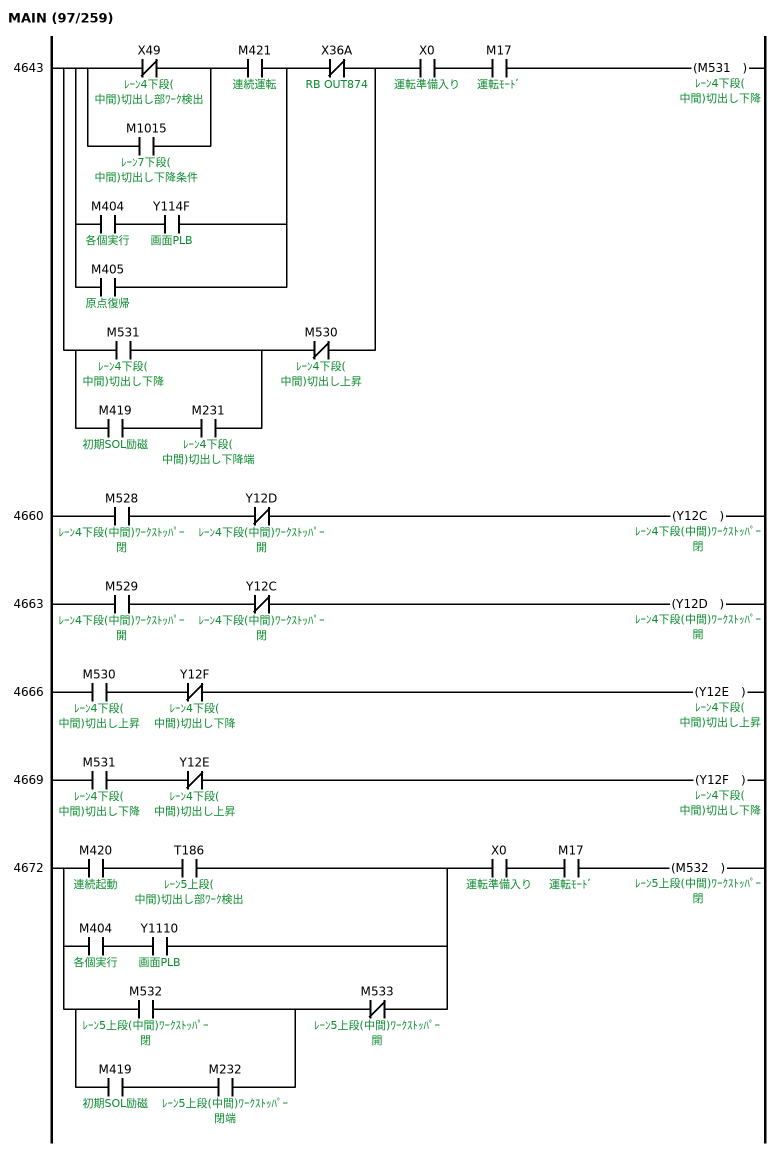
[picture p96: ladder of MAIN, rungs at steps 4643 to 4672]
4643  LDI     X49  ; ﾚｰﾝ4下段(中間)切出し部ﾜｰｸ検出
      OR      M1015  ; ﾚｰﾝ7下段(中間)切出し下降条件
      AND     M421  ; 連続運転
      LD      M404  ; 各個実行
      AND     Y114F  ; 画面PLB
      ORB
      OR      M405  ; 原点復帰
      ANI     X36A  ; RB OUT874
      LD      M531  ; ﾚｰﾝ4下段(中間)切出し下降
      LD      M419  ; 初期SOL励磁
      AND     M231  ; ﾚｰﾝ4下段(中間)切出し下降端
      ORB
      ANI     M530  ; ﾚｰﾝ4下段(中間)切出し上昇
      ORB
      AND     X0  ; 運転準備入り
      AND     M17  ; 運転ﾓｰﾄﾞ
      OUT     M531  ; ﾚｰﾝ4下段(中間)切出し下降
4660  LD      M528  ; ﾚｰﾝ4下段(中間)ﾜｰｸｽﾄｯﾊﾟｰ閉
      ANI     Y12D  ; ﾚｰﾝ4下段(中間)ﾜｰｸｽﾄｯﾊﾟｰ開
      OUT     Y12C  ; ﾚｰﾝ4下段(中間)ﾜｰｸｽﾄｯﾊﾟｰ閉
4663  LD      M529  ; ﾚｰﾝ4下段(中間)ﾜｰｸｽﾄｯﾊﾟｰ開
      ANI     Y12C  ; ﾚｰﾝ4下段(中間)ﾜｰｸｽﾄｯﾊﾟｰ閉
      OUT     Y12D  ; ﾚｰﾝ4下段(中間)ﾜｰｸｽﾄｯﾊﾟｰ開
4666  LD      M530  ; ﾚｰﾝ4下段(中間)切出し上昇
      ANI     Y12F  ; ﾚｰﾝ4下段(中間)切出し下降
      OUT     Y12E  ; ﾚｰﾝ4下段(中間)切出し上昇
4669  LD      M531  ; ﾚｰﾝ4下段(中間)切出し下降
      ANI     Y12E  ; ﾚｰﾝ4下段(中間)切出し上昇
      OUT     Y12F  ; ﾚｰﾝ4下段(中間)切出し下降
4672  LD      M420  ; 連続起動
      AND     T186  ; ﾚｰﾝ5上段(中間)切出し部ﾜｰｸ検出
      LD      M404  ; 各個実行
      AND     Y1110  ; 画面PLB
      ORB
      LD      M532  ; ﾚｰﾝ5上段(中間)ﾜｰｸｽﾄｯﾊﾟｰ閉
      LD      M419  ; 初期SOL励磁
      AND     M232  ; ﾚｰﾝ5上段(中間)ﾜｰｸｽﾄｯﾊﾟｰ閉端
      ORB
      ANI     M533  ; ﾚｰﾝ5上段(中間)ﾜｰｸｽﾄｯﾊﾟｰ開
      ORB
      AND     X0  ; 運転準備入り
      AND     M17  ; 運転ﾓｰﾄﾞ
      OUT     M532  ; ﾚｰﾝ5上段(中間)ﾜｰｸｽﾄｯﾊﾟｰ閉
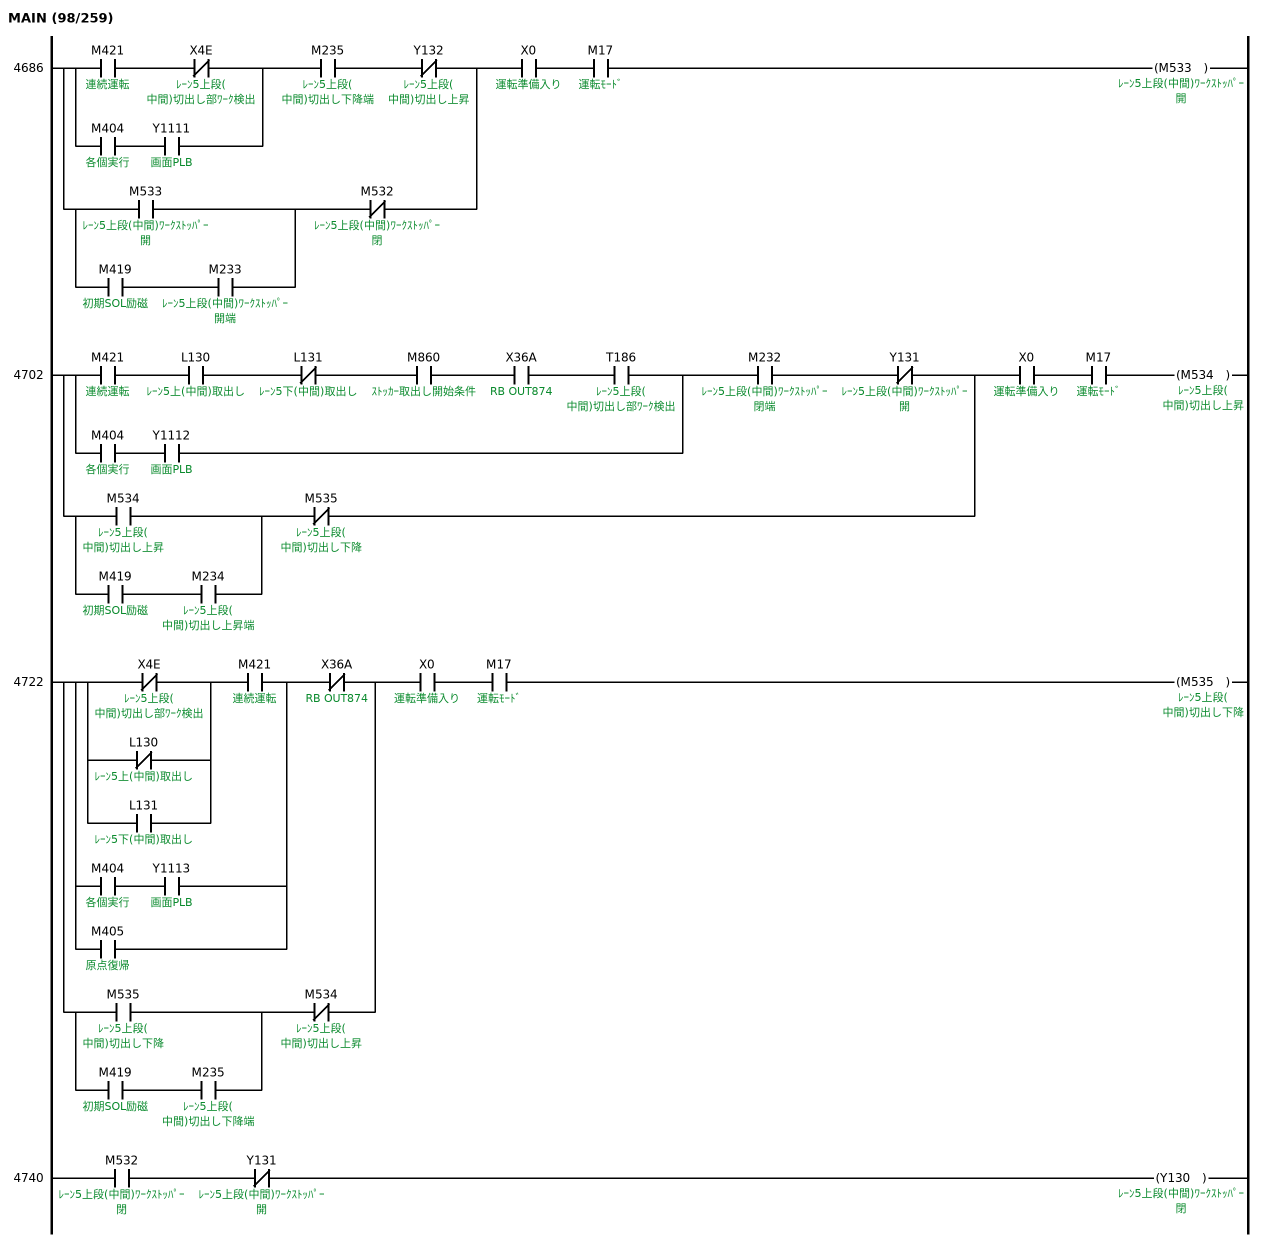
4686  LD      M421  ; 連続運転
      ANI     X4E  ; ﾚｰﾝ5上段(中間)切出し部ﾜｰｸ検出
      LD      M404  ; 各個実行
      AND     Y1111  ; 画面PLB
      ORB
      AND     M235  ; ﾚｰﾝ5上段(中間)切出し下降端
      ANI     Y132  ; ﾚｰﾝ5上段(中間)切出し上昇
      LD      M533  ; ﾚｰﾝ5上段(中間)ﾜｰｸｽﾄｯﾊﾟｰ開
      LD      M419  ; 初期SOL励磁
      AND     M233  ; ﾚｰﾝ5上段(中間)ﾜｰｸｽﾄｯﾊﾟｰ開端
      ORB
      ANI     M532  ; ﾚｰﾝ5上段(中間)ﾜｰｸｽﾄｯﾊﾟｰ閉
      ORB
      AND     X0  ; 運転準備入り
      AND     M17  ; 運転ﾓｰﾄﾞ
      OUT     M533  ; ﾚｰﾝ5上段(中間)ﾜｰｸｽﾄｯﾊﾟｰ開
4702  LD      M421  ; 連続運転
      AND     L130  ; ﾚｰﾝ5上(中間)取出し
      ANI     L131  ; ﾚｰﾝ5下(中間)取出し
      AND     M860  ; ｽﾄｯｶｰ取出し開始条件
      AND     X36A  ; RB OUT874
      AND     T186  ; ﾚｰﾝ5上段(中間)切出し部ﾜｰｸ検出
      LD      M404  ; 各個実行
      AND     Y1112  ; 画面PLB
      ORB
      AND     M232  ; ﾚｰﾝ5上段(中間)ﾜｰｸｽﾄｯﾊﾟｰ閉端
      ANI     Y131  ; ﾚｰﾝ5上段(中間)ﾜｰｸｽﾄｯﾊﾟｰ開
      LD      M534  ; ﾚｰﾝ5上段(中間)切出し上昇
      LD      M419  ; 初期SOL励磁
      AND     M234  ; ﾚｰﾝ5上段(中間)切出し上昇端
      ORB
      ANI     M535  ; ﾚｰﾝ5上段(中間)切出し下降
      ORB
      AND     X0  ; 運転準備入り
      AND     M17  ; 運転ﾓｰﾄﾞ
      OUT     M534  ; ﾚｰﾝ5上段(中間)切出し上昇
4722  LDI     X4E  ; ﾚｰﾝ5上段(中間)切出し部ﾜｰｸ検出
      ORI     L130  ; ﾚｰﾝ5上(中間)取出し
      OR      L131  ; ﾚｰﾝ5下(中間)取出し
      AND     M421  ; 連続運転
      LD      M404  ; 各個実行
      AND     Y1113  ; 画面PLB
      ORB
      OR      M405  ; 原点復帰
      ANI     X36A  ; RB OUT874
      LD      M535  ; ﾚｰﾝ5上段(中間)切出し下降
      LD      M419  ; 初期SOL励磁
      AND     M235  ; ﾚｰﾝ5上段(中間)切出し下降端
      ORB
      ANI     M534  ; ﾚｰﾝ5上段(中間)切出し上昇
      ORB
      AND     X0  ; 運転準備入り
      AND     M17  ; 運転ﾓｰﾄﾞ
      OUT     M535  ; ﾚｰﾝ5上段(中間)切出し下降
4740  LD      M532  ; ﾚｰﾝ5上段(中間)ﾜｰｸｽﾄｯﾊﾟｰ閉
      ANI     Y131  ; ﾚｰﾝ5上段(中間)ﾜｰｸｽﾄｯﾊﾟｰ開
      OUT     Y130  ; ﾚｰﾝ5上段(中間)ﾜｰｸｽﾄｯﾊﾟｰ閉
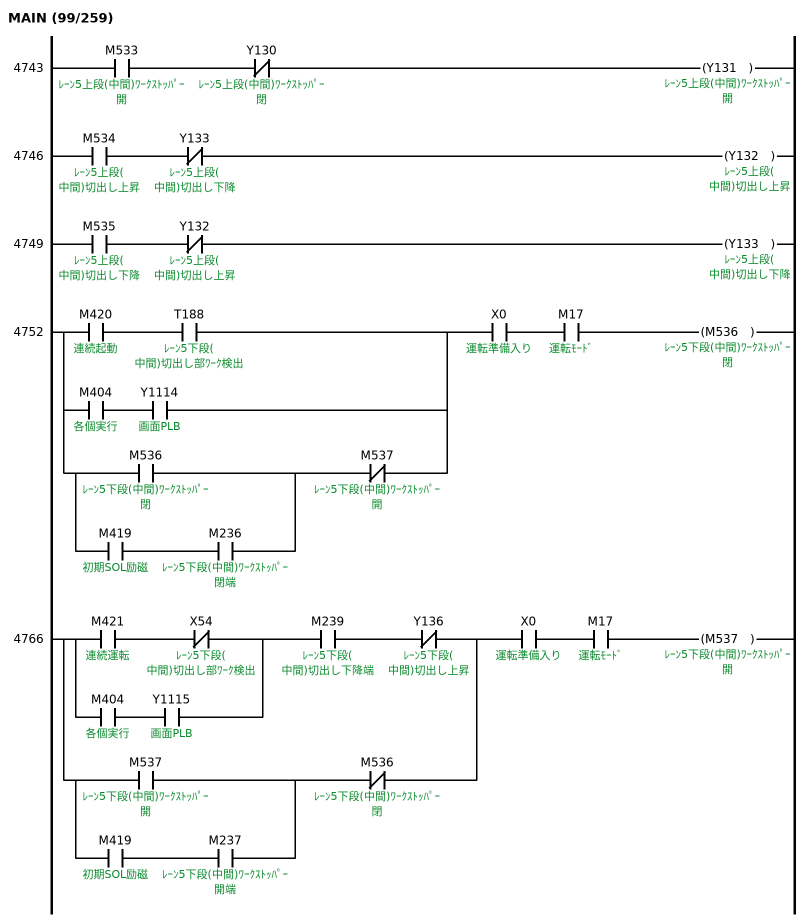
4743  LD      M533  ; ﾚｰﾝ5上段(中間)ﾜｰｸｽﾄｯﾊﾟｰ開
      ANI     Y130  ; ﾚｰﾝ5上段(中間)ﾜｰｸｽﾄｯﾊﾟｰ閉
      OUT     Y131  ; ﾚｰﾝ5上段(中間)ﾜｰｸｽﾄｯﾊﾟｰ開
4746  LD      M534  ; ﾚｰﾝ5上段(中間)切出し上昇
      ANI     Y133  ; ﾚｰﾝ5上段(中間)切出し下降
      OUT     Y132  ; ﾚｰﾝ5上段(中間)切出し上昇
4749  LD      M535  ; ﾚｰﾝ5上段(中間)切出し下降
      ANI     Y132  ; ﾚｰﾝ5上段(中間)切出し上昇
      OUT     Y133  ; ﾚｰﾝ5上段(中間)切出し下降
4752  LD      M420  ; 連続起動
      AND     T188  ; ﾚｰﾝ5下段(中間)切出し部ﾜｰｸ検出
      LD      M404  ; 各個実行
      AND     Y1114  ; 画面PLB
      ORB
      LD      M536  ; ﾚｰﾝ5下段(中間)ﾜｰｸｽﾄｯﾊﾟｰ閉
      LD      M419  ; 初期SOL励磁
      AND     M236  ; ﾚｰﾝ5下段(中間)ﾜｰｸｽﾄｯﾊﾟｰ閉端
      ORB
      ANI     M537  ; ﾚｰﾝ5下段(中間)ﾜｰｸｽﾄｯﾊﾟｰ開
      ORB
      AND     X0  ; 運転準備入り
      AND     M17  ; 運転ﾓｰﾄﾞ
      OUT     M536  ; ﾚｰﾝ5下段(中間)ﾜｰｸｽﾄｯﾊﾟｰ閉
4766  LD      M421  ; 連続運転
      ANI     X54  ; ﾚｰﾝ5下段(中間)切出し部ﾜｰｸ検出
      LD      M404  ; 各個実行
      AND     Y1115  ; 画面PLB
      ORB
      AND     M239  ; ﾚｰﾝ5下段(中間)切出し下降端
      ANI     Y136  ; ﾚｰﾝ5下段(中間)切出し上昇
      LD      M537  ; ﾚｰﾝ5下段(中間)ﾜｰｸｽﾄｯﾊﾟｰ開
      LD      M419  ; 初期SOL励磁
      AND     M237  ; ﾚｰﾝ5下段(中間)ﾜｰｸｽﾄｯﾊﾟｰ開端
      ORB
      ANI     M536  ; ﾚｰﾝ5下段(中間)ﾜｰｸｽﾄｯﾊﾟｰ閉
      ORB
      AND     X0  ; 運転準備入り
      AND     M17  ; 運転ﾓｰﾄﾞ
      OUT     M537  ; ﾚｰﾝ5下段(中間)ﾜｰｸｽﾄｯﾊﾟｰ開
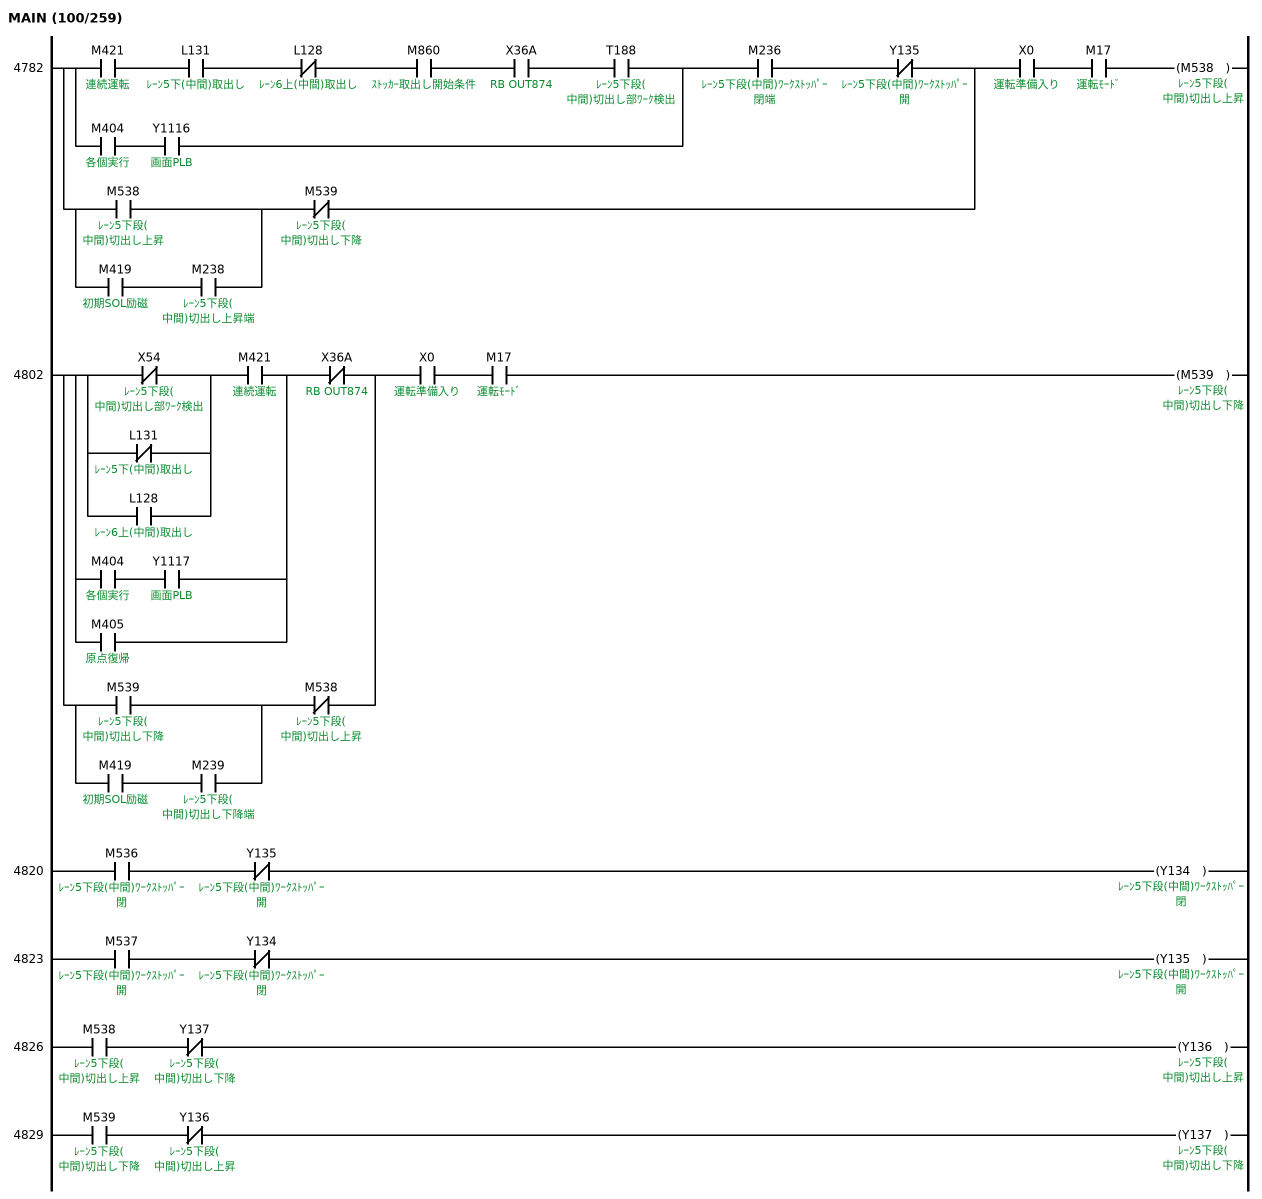
4782  LD      M421  ; 連続運転
      AND     L131  ; ﾚｰﾝ5下(中間)取出し
      ANI     L128  ; ﾚｰﾝ6上(中間)取出し
      AND     M860  ; ｽﾄｯｶｰ取出し開始条件
      AND     X36A  ; RB OUT874
      AND     T188  ; ﾚｰﾝ5下段(中間)切出し部ﾜｰｸ検出
      LD      M404  ; 各個実行
      AND     Y1116  ; 画面PLB
      ORB
      AND     M236  ; ﾚｰﾝ5下段(中間)ﾜｰｸｽﾄｯﾊﾟｰ閉端
      ANI     Y135  ; ﾚｰﾝ5下段(中間)ﾜｰｸｽﾄｯﾊﾟｰ開
      LD      M538  ; ﾚｰﾝ5下段(中間)切出し上昇
      LD      M419  ; 初期SOL励磁
      AND     M238  ; ﾚｰﾝ5下段(中間)切出し上昇端
      ORB
      ANI     M539  ; ﾚｰﾝ5下段(中間)切出し下降
      ORB
      AND     X0  ; 運転準備入り
      AND     M17  ; 運転ﾓｰﾄﾞ
      OUT     M538  ; ﾚｰﾝ5下段(中間)切出し上昇
4802  LDI     X54  ; ﾚｰﾝ5下段(中間)切出し部ﾜｰｸ検出
      ORI     L131  ; ﾚｰﾝ5下(中間)取出し
      OR      L128  ; ﾚｰﾝ6上(中間)取出し
      AND     M421  ; 連続運転
      LD      M404  ; 各個実行
      AND     Y1117  ; 画面PLB
      ORB
      OR      M405  ; 原点復帰
      ANI     X36A  ; RB OUT874
      LD      M539  ; ﾚｰﾝ5下段(中間)切出し下降
      LD      M419  ; 初期SOL励磁
      AND     M239  ; ﾚｰﾝ5下段(中間)切出し下降端
      ORB
      ANI     M538  ; ﾚｰﾝ5下段(中間)切出し上昇
      ORB
      AND     X0  ; 運転準備入り
      AND     M17  ; 運転ﾓｰﾄﾞ
      OUT     M539  ; ﾚｰﾝ5下段(中間)切出し下降
4820  LD      M536  ; ﾚｰﾝ5下段(中間)ﾜｰｸｽﾄｯﾊﾟｰ閉
      ANI     Y135  ; ﾚｰﾝ5下段(中間)ﾜｰｸｽﾄｯﾊﾟｰ開
      OUT     Y134  ; ﾚｰﾝ5下段(中間)ﾜｰｸｽﾄｯﾊﾟｰ閉
4823  LD      M537  ; ﾚｰﾝ5下段(中間)ﾜｰｸｽﾄｯﾊﾟｰ開
      ANI     Y134  ; ﾚｰﾝ5下段(中間)ﾜｰｸｽﾄｯﾊﾟｰ閉
      OUT     Y135  ; ﾚｰﾝ5下段(中間)ﾜｰｸｽﾄｯﾊﾟｰ開
4826  LD      M538  ; ﾚｰﾝ5下段(中間)切出し上昇
      ANI     Y137  ; ﾚｰﾝ5下段(中間)切出し下降
      OUT     Y136  ; ﾚｰﾝ5下段(中間)切出し上昇
4829  LD      M539  ; ﾚｰﾝ5下段(中間)切出し下降
      ANI     Y136  ; ﾚｰﾝ5下段(中間)切出し上昇
      OUT     Y137  ; ﾚｰﾝ5下段(中間)切出し下降
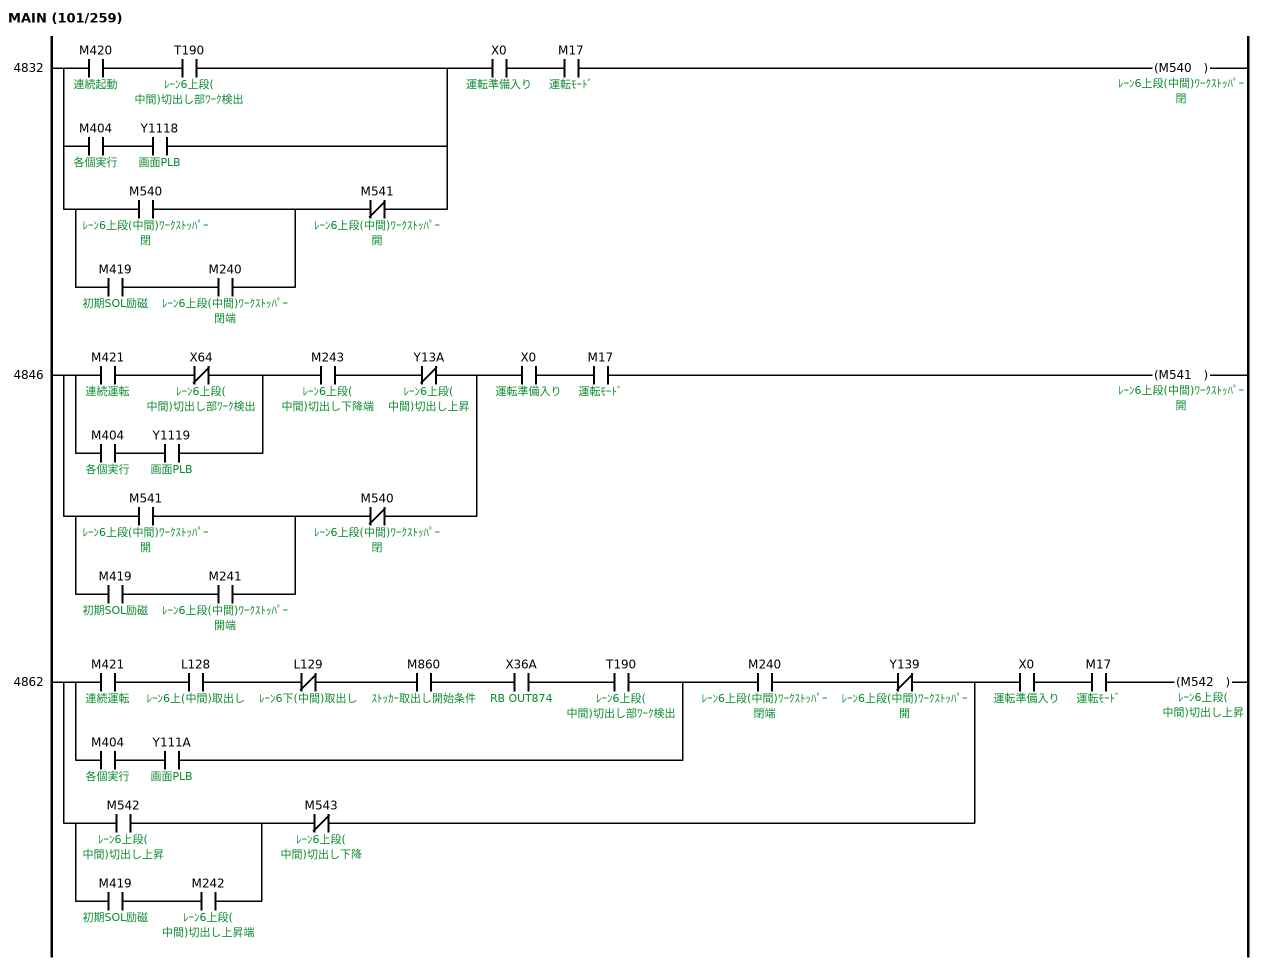
4832  LD      M420  ; 連続起動
      AND     T190  ; ﾚｰﾝ6上段(中間)切出し部ﾜｰｸ検出
      LD      M404  ; 各個実行
      AND     Y1118  ; 画面PLB
      ORB
      LD      M540  ; ﾚｰﾝ6上段(中間)ﾜｰｸｽﾄｯﾊﾟｰ閉
      LD      M419  ; 初期SOL励磁
      AND     M240  ; ﾚｰﾝ6上段(中間)ﾜｰｸｽﾄｯﾊﾟｰ閉端
      ORB
      ANI     M541  ; ﾚｰﾝ6上段(中間)ﾜｰｸｽﾄｯﾊﾟｰ開
      ORB
      AND     X0  ; 運転準備入り
      AND     M17  ; 運転ﾓｰﾄﾞ
      OUT     M540  ; ﾚｰﾝ6上段(中間)ﾜｰｸｽﾄｯﾊﾟｰ閉
4846  LD      M421  ; 連続運転
      ANI     X64  ; ﾚｰﾝ6上段(中間)切出し部ﾜｰｸ検出
      LD      M404  ; 各個実行
      AND     Y1119  ; 画面PLB
      ORB
      AND     M243  ; ﾚｰﾝ6上段(中間)切出し下降端
      ANI     Y13A  ; ﾚｰﾝ6上段(中間)切出し上昇
      LD      M541  ; ﾚｰﾝ6上段(中間)ﾜｰｸｽﾄｯﾊﾟｰ開
      LD      M419  ; 初期SOL励磁
      AND     M241  ; ﾚｰﾝ6上段(中間)ﾜｰｸｽﾄｯﾊﾟｰ開端
      ORB
      ANI     M540  ; ﾚｰﾝ6上段(中間)ﾜｰｸｽﾄｯﾊﾟｰ閉
      ORB
      AND     X0  ; 運転準備入り
      AND     M17  ; 運転ﾓｰﾄﾞ
      OUT     M541  ; ﾚｰﾝ6上段(中間)ﾜｰｸｽﾄｯﾊﾟｰ開
4862  LD      M421  ; 連続運転
      AND     L128  ; ﾚｰﾝ6上(中間)取出し
      ANI     L129  ; ﾚｰﾝ6下(中間)取出し
      AND     M860  ; ｽﾄｯｶｰ取出し開始条件
      AND     X36A  ; RB OUT874
      AND     T190  ; ﾚｰﾝ6上段(中間)切出し部ﾜｰｸ検出
      LD      M404  ; 各個実行
      AND     Y111A  ; 画面PLB
      ORB
      AND     M240  ; ﾚｰﾝ6上段(中間)ﾜｰｸｽﾄｯﾊﾟｰ閉端
      ANI     Y139  ; ﾚｰﾝ6上段(中間)ﾜｰｸｽﾄｯﾊﾟｰ開
      LD      M542  ; ﾚｰﾝ6上段(中間)切出し上昇
      LD      M419  ; 初期SOL励磁
      AND     M242  ; ﾚｰﾝ6上段(中間)切出し上昇端
      ORB
      ANI     M543  ; ﾚｰﾝ6上段(中間)切出し下降
      ORB
      AND     X0  ; 運転準備入り
      AND     M17  ; 運転ﾓｰﾄﾞ
      OUT     M542  ; ﾚｰﾝ6上段(中間)切出し上昇
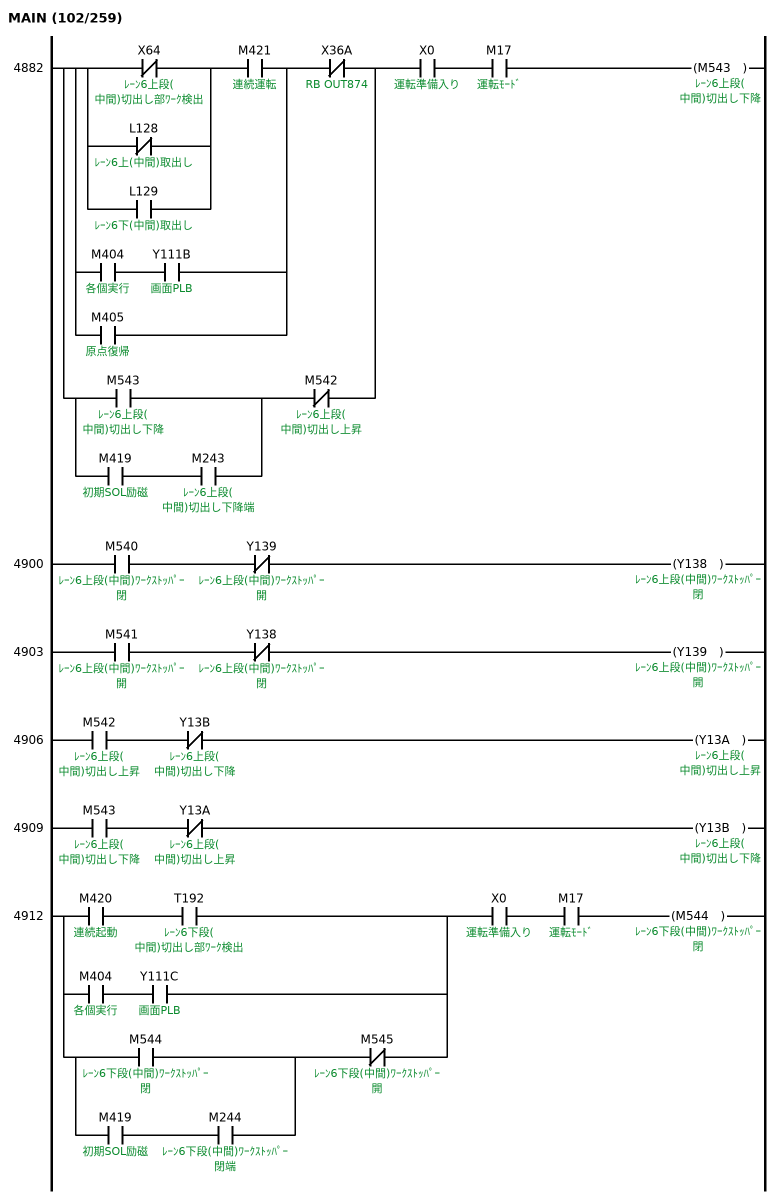
4882  LDI     X64  ; ﾚｰﾝ6上段(中間)切出し部ﾜｰｸ検出
      ORI     L128  ; ﾚｰﾝ6上(中間)取出し
      OR      L129  ; ﾚｰﾝ6下(中間)取出し
      AND     M421  ; 連続運転
      LD      M404  ; 各個実行
      AND     Y111B  ; 画面PLB
      ORB
      OR      M405  ; 原点復帰
      ANI     X36A  ; RB OUT874
      LD      M543  ; ﾚｰﾝ6上段(中間)切出し下降
      LD      M419  ; 初期SOL励磁
      AND     M243  ; ﾚｰﾝ6上段(中間)切出し下降端
      ORB
      ANI     M542  ; ﾚｰﾝ6上段(中間)切出し上昇
      ORB
      AND     X0  ; 運転準備入り
      AND     M17  ; 運転ﾓｰﾄﾞ
      OUT     M543  ; ﾚｰﾝ6上段(中間)切出し下降
4900  LD      M540  ; ﾚｰﾝ6上段(中間)ﾜｰｸｽﾄｯﾊﾟｰ閉
      ANI     Y139  ; ﾚｰﾝ6上段(中間)ﾜｰｸｽﾄｯﾊﾟｰ開
      OUT     Y138  ; ﾚｰﾝ6上段(中間)ﾜｰｸｽﾄｯﾊﾟｰ閉
4903  LD      M541  ; ﾚｰﾝ6上段(中間)ﾜｰｸｽﾄｯﾊﾟｰ開
      ANI     Y138  ; ﾚｰﾝ6上段(中間)ﾜｰｸｽﾄｯﾊﾟｰ閉
      OUT     Y139  ; ﾚｰﾝ6上段(中間)ﾜｰｸｽﾄｯﾊﾟｰ開
4906  LD      M542  ; ﾚｰﾝ6上段(中間)切出し上昇
      ANI     Y13B  ; ﾚｰﾝ6上段(中間)切出し下降
      OUT     Y13A  ; ﾚｰﾝ6上段(中間)切出し上昇
4909  LD      M543  ; ﾚｰﾝ6上段(中間)切出し下降
      ANI     Y13A  ; ﾚｰﾝ6上段(中間)切出し上昇
      OUT     Y13B  ; ﾚｰﾝ6上段(中間)切出し下降
4912  LD      M420  ; 連続起動
      AND     T192  ; ﾚｰﾝ6下段(中間)切出し部ﾜｰｸ検出
      LD      M404  ; 各個実行
      AND     Y111C  ; 画面PLB
      ORB
      LD      M544  ; ﾚｰﾝ6下段(中間)ﾜｰｸｽﾄｯﾊﾟｰ閉
      LD      M419  ; 初期SOL励磁
      AND     M244  ; ﾚｰﾝ6下段(中間)ﾜｰｸｽﾄｯﾊﾟｰ閉端
      ORB
      ANI     M545  ; ﾚｰﾝ6下段(中間)ﾜｰｸｽﾄｯﾊﾟｰ開
      ORB
      AND     X0  ; 運転準備入り
      AND     M17  ; 運転ﾓｰﾄﾞ
      OUT     M544  ; ﾚｰﾝ6下段(中間)ﾜｰｸｽﾄｯﾊﾟｰ閉
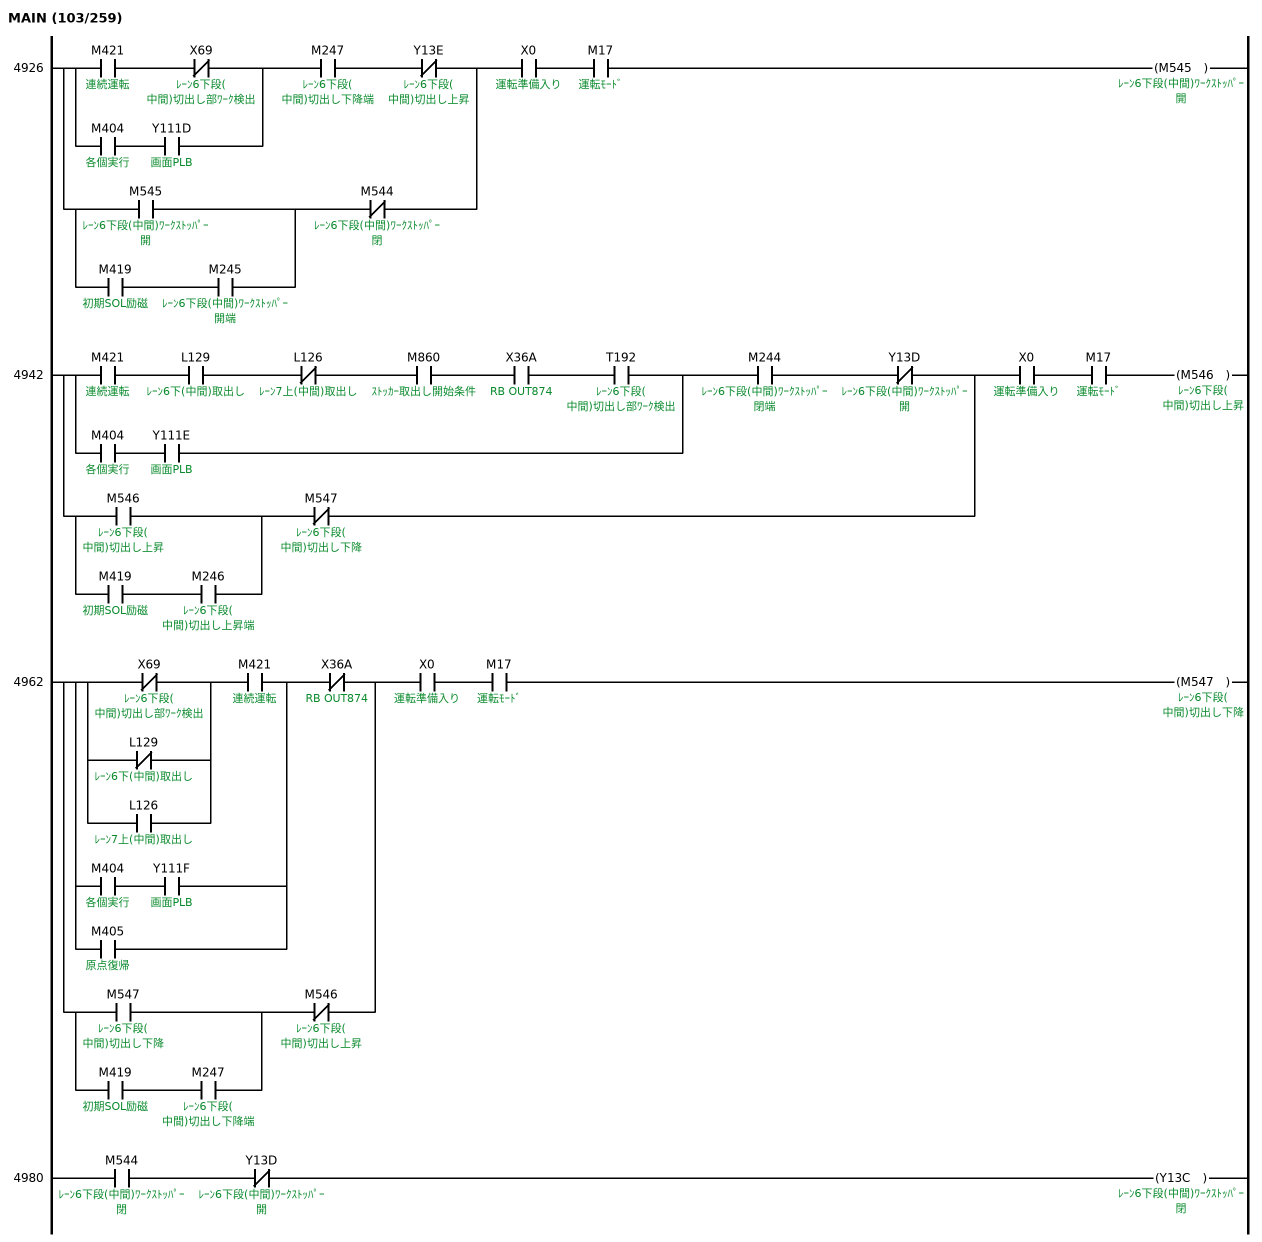
4926  LD      M421  ; 連続運転
      ANI     X69  ; ﾚｰﾝ6下段(中間)切出し部ﾜｰｸ検出
      LD      M404  ; 各個実行
      AND     Y111D  ; 画面PLB
      ORB
      AND     M247  ; ﾚｰﾝ6下段(中間)切出し下降端
      ANI     Y13E  ; ﾚｰﾝ6下段(中間)切出し上昇
      LD      M545  ; ﾚｰﾝ6下段(中間)ﾜｰｸｽﾄｯﾊﾟｰ開
      LD      M419  ; 初期SOL励磁
      AND     M245  ; ﾚｰﾝ6下段(中間)ﾜｰｸｽﾄｯﾊﾟｰ開端
      ORB
      ANI     M544  ; ﾚｰﾝ6下段(中間)ﾜｰｸｽﾄｯﾊﾟｰ閉
      ORB
      AND     X0  ; 運転準備入り
      AND     M17  ; 運転ﾓｰﾄﾞ
      OUT     M545  ; ﾚｰﾝ6下段(中間)ﾜｰｸｽﾄｯﾊﾟｰ開
4942  LD      M421  ; 連続運転
      AND     L129  ; ﾚｰﾝ6下(中間)取出し
      ANI     L126  ; ﾚｰﾝ7上(中間)取出し
      AND     M860  ; ｽﾄｯｶｰ取出し開始条件
      AND     X36A  ; RB OUT874
      AND     T192  ; ﾚｰﾝ6下段(中間)切出し部ﾜｰｸ検出
      LD      M404  ; 各個実行
      AND     Y111E  ; 画面PLB
      ORB
      AND     M244  ; ﾚｰﾝ6下段(中間)ﾜｰｸｽﾄｯﾊﾟｰ閉端
      ANI     Y13D  ; ﾚｰﾝ6下段(中間)ﾜｰｸｽﾄｯﾊﾟｰ開
      LD      M546  ; ﾚｰﾝ6下段(中間)切出し上昇
      LD      M419  ; 初期SOL励磁
      AND     M246  ; ﾚｰﾝ6下段(中間)切出し上昇端
      ORB
      ANI     M547  ; ﾚｰﾝ6下段(中間)切出し下降
      ORB
      AND     X0  ; 運転準備入り
      AND     M17  ; 運転ﾓｰﾄﾞ
      OUT     M546  ; ﾚｰﾝ6下段(中間)切出し上昇
4962  LDI     X69  ; ﾚｰﾝ6下段(中間)切出し部ﾜｰｸ検出
      ORI     L129  ; ﾚｰﾝ6下(中間)取出し
      OR      L126  ; ﾚｰﾝ7上(中間)取出し
      AND     M421  ; 連続運転
      LD      M404  ; 各個実行
      AND     Y111F  ; 画面PLB
      ORB
      OR      M405  ; 原点復帰
      ANI     X36A  ; RB OUT874
      LD      M547  ; ﾚｰﾝ6下段(中間)切出し下降
      LD      M419  ; 初期SOL励磁
      AND     M247  ; ﾚｰﾝ6下段(中間)切出し下降端
      ORB
      ANI     M546  ; ﾚｰﾝ6下段(中間)切出し上昇
      ORB
      AND     X0  ; 運転準備入り
      AND     M17  ; 運転ﾓｰﾄﾞ
      OUT     M547  ; ﾚｰﾝ6下段(中間)切出し下降
4980  LD      M544  ; ﾚｰﾝ6下段(中間)ﾜｰｸｽﾄｯﾊﾟｰ閉
      ANI     Y13D  ; ﾚｰﾝ6下段(中間)ﾜｰｸｽﾄｯﾊﾟｰ開
      OUT     Y13C  ; ﾚｰﾝ6下段(中間)ﾜｰｸｽﾄｯﾊﾟｰ閉
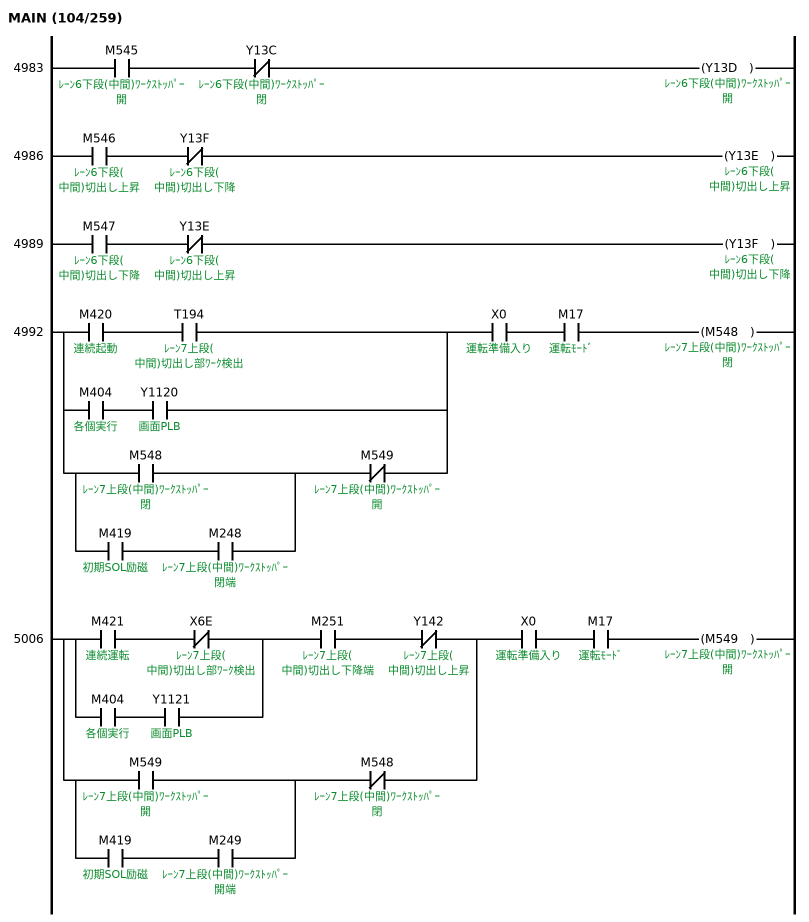
4983  LD      M545  ; ﾚｰﾝ6下段(中間)ﾜｰｸｽﾄｯﾊﾟｰ開
      ANI     Y13C  ; ﾚｰﾝ6下段(中間)ﾜｰｸｽﾄｯﾊﾟｰ閉
      OUT     Y13D  ; ﾚｰﾝ6下段(中間)ﾜｰｸｽﾄｯﾊﾟｰ開
4986  LD      M546  ; ﾚｰﾝ6下段(中間)切出し上昇
      ANI     Y13F  ; ﾚｰﾝ6下段(中間)切出し下降
      OUT     Y13E  ; ﾚｰﾝ6下段(中間)切出し上昇
4989  LD      M547  ; ﾚｰﾝ6下段(中間)切出し下降
      ANI     Y13E  ; ﾚｰﾝ6下段(中間)切出し上昇
      OUT     Y13F  ; ﾚｰﾝ6下段(中間)切出し下降
4992  LD      M420  ; 連続起動
      AND     T194  ; ﾚｰﾝ7上段(中間)切出し部ﾜｰｸ検出
      LD      M404  ; 各個実行
      AND     Y1120  ; 画面PLB
      ORB
      LD      M548  ; ﾚｰﾝ7上段(中間)ﾜｰｸｽﾄｯﾊﾟｰ閉
      LD      M419  ; 初期SOL励磁
      AND     M248  ; ﾚｰﾝ7上段(中間)ﾜｰｸｽﾄｯﾊﾟｰ閉端
      ORB
      ANI     M549  ; ﾚｰﾝ7上段(中間)ﾜｰｸｽﾄｯﾊﾟｰ開
      ORB
      AND     X0  ; 運転準備入り
      AND     M17  ; 運転ﾓｰﾄﾞ
      OUT     M548  ; ﾚｰﾝ7上段(中間)ﾜｰｸｽﾄｯﾊﾟｰ閉
5006  LD      M421  ; 連続運転
      ANI     X6E  ; ﾚｰﾝ7上段(中間)切出し部ﾜｰｸ検出
      LD      M404  ; 各個実行
      AND     Y1121  ; 画面PLB
      ORB
      AND     M251  ; ﾚｰﾝ7上段(中間)切出し下降端
      ANI     Y142  ; ﾚｰﾝ7上段(中間)切出し上昇
      LD      M549  ; ﾚｰﾝ7上段(中間)ﾜｰｸｽﾄｯﾊﾟｰ開
      LD      M419  ; 初期SOL励磁
      AND     M249  ; ﾚｰﾝ7上段(中間)ﾜｰｸｽﾄｯﾊﾟｰ開端
      ORB
      ANI     M548  ; ﾚｰﾝ7上段(中間)ﾜｰｸｽﾄｯﾊﾟｰ閉
      ORB
      AND     X0  ; 運転準備入り
      AND     M17  ; 運転ﾓｰﾄﾞ
      OUT     M549  ; ﾚｰﾝ7上段(中間)ﾜｰｸｽﾄｯﾊﾟｰ開
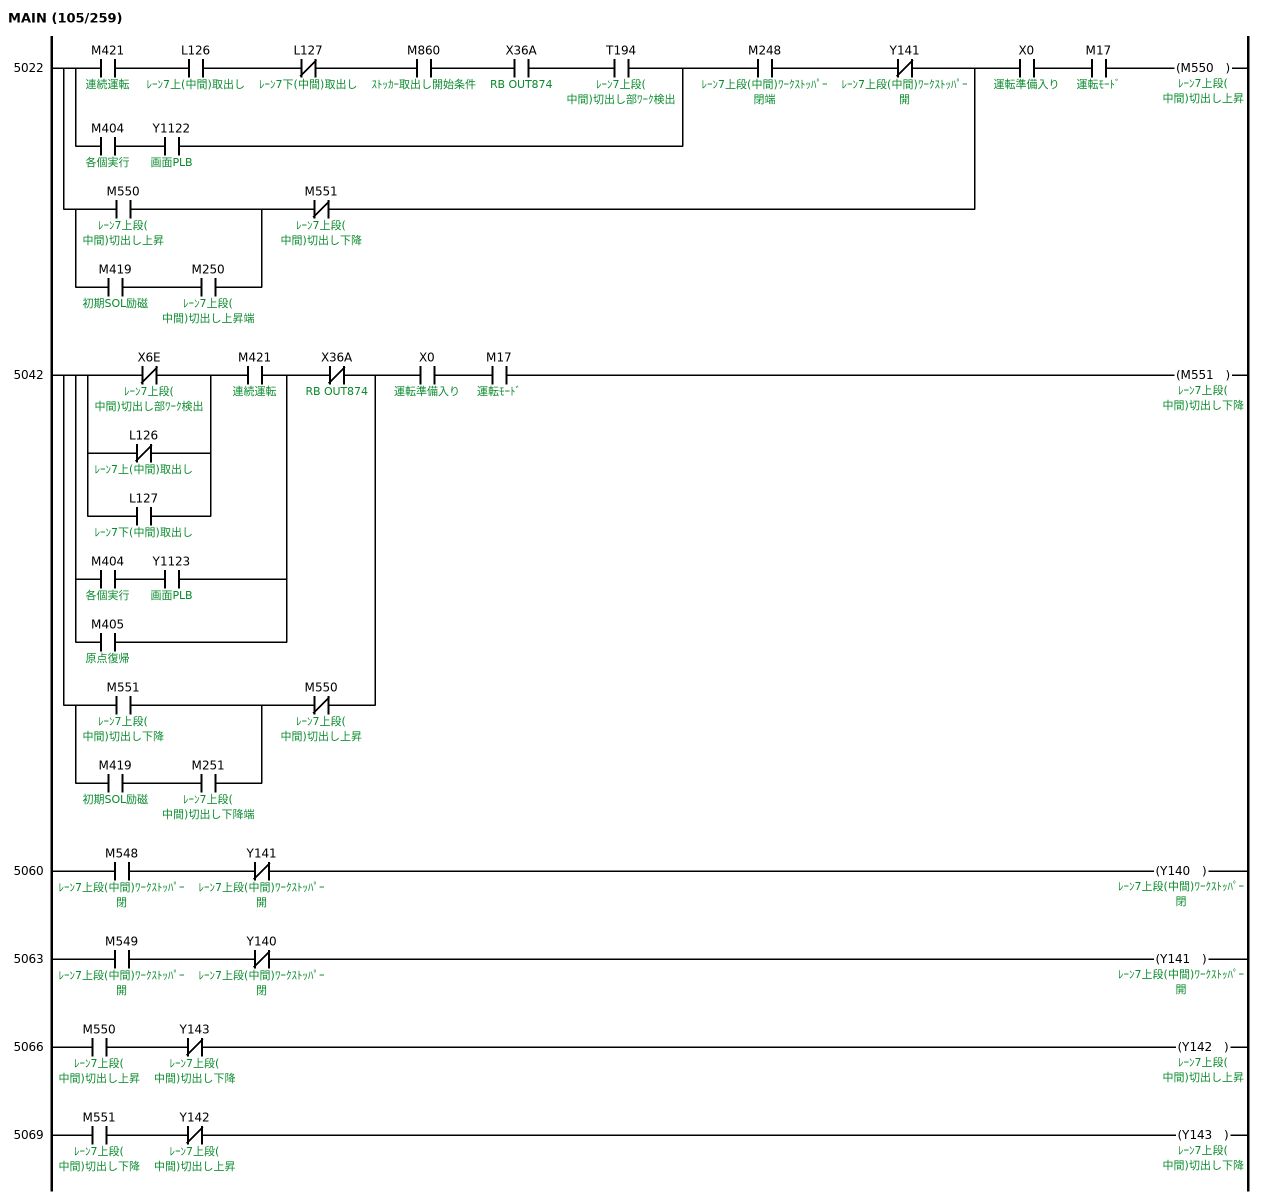
5022  LD      M421  ; 連続運転
      AND     L126  ; ﾚｰﾝ7上(中間)取出し
      ANI     L127  ; ﾚｰﾝ7下(中間)取出し
      AND     M860  ; ｽﾄｯｶｰ取出し開始条件
      AND     X36A  ; RB OUT874
      AND     T194  ; ﾚｰﾝ7上段(中間)切出し部ﾜｰｸ検出
      LD      M404  ; 各個実行
      AND     Y1122  ; 画面PLB
      ORB
      AND     M248  ; ﾚｰﾝ7上段(中間)ﾜｰｸｽﾄｯﾊﾟｰ閉端
      ANI     Y141  ; ﾚｰﾝ7上段(中間)ﾜｰｸｽﾄｯﾊﾟｰ開
      LD      M550  ; ﾚｰﾝ7上段(中間)切出し上昇
      LD      M419  ; 初期SOL励磁
      AND     M250  ; ﾚｰﾝ7上段(中間)切出し上昇端
      ORB
      ANI     M551  ; ﾚｰﾝ7上段(中間)切出し下降
      ORB
      AND     X0  ; 運転準備入り
      AND     M17  ; 運転ﾓｰﾄﾞ
      OUT     M550  ; ﾚｰﾝ7上段(中間)切出し上昇
5042  LDI     X6E  ; ﾚｰﾝ7上段(中間)切出し部ﾜｰｸ検出
      ORI     L126  ; ﾚｰﾝ7上(中間)取出し
      OR      L127  ; ﾚｰﾝ7下(中間)取出し
      AND     M421  ; 連続運転
      LD      M404  ; 各個実行
      AND     Y1123  ; 画面PLB
      ORB
      OR      M405  ; 原点復帰
      ANI     X36A  ; RB OUT874
      LD      M551  ; ﾚｰﾝ7上段(中間)切出し下降
      LD      M419  ; 初期SOL励磁
      AND     M251  ; ﾚｰﾝ7上段(中間)切出し下降端
      ORB
      ANI     M550  ; ﾚｰﾝ7上段(中間)切出し上昇
      ORB
      AND     X0  ; 運転準備入り
      AND     M17  ; 運転ﾓｰﾄﾞ
      OUT     M551  ; ﾚｰﾝ7上段(中間)切出し下降
5060  LD      M548  ; ﾚｰﾝ7上段(中間)ﾜｰｸｽﾄｯﾊﾟｰ閉
      ANI     Y141  ; ﾚｰﾝ7上段(中間)ﾜｰｸｽﾄｯﾊﾟｰ開
      OUT     Y140  ; ﾚｰﾝ7上段(中間)ﾜｰｸｽﾄｯﾊﾟｰ閉
5063  LD      M549  ; ﾚｰﾝ7上段(中間)ﾜｰｸｽﾄｯﾊﾟｰ開
      ANI     Y140  ; ﾚｰﾝ7上段(中間)ﾜｰｸｽﾄｯﾊﾟｰ閉
      OUT     Y141  ; ﾚｰﾝ7上段(中間)ﾜｰｸｽﾄｯﾊﾟｰ開
5066  LD      M550  ; ﾚｰﾝ7上段(中間)切出し上昇
      ANI     Y143  ; ﾚｰﾝ7上段(中間)切出し下降
      OUT     Y142  ; ﾚｰﾝ7上段(中間)切出し上昇
5069  LD      M551  ; ﾚｰﾝ7上段(中間)切出し下降
      ANI     Y142  ; ﾚｰﾝ7上段(中間)切出し上昇
      OUT     Y143  ; ﾚｰﾝ7上段(中間)切出し下降
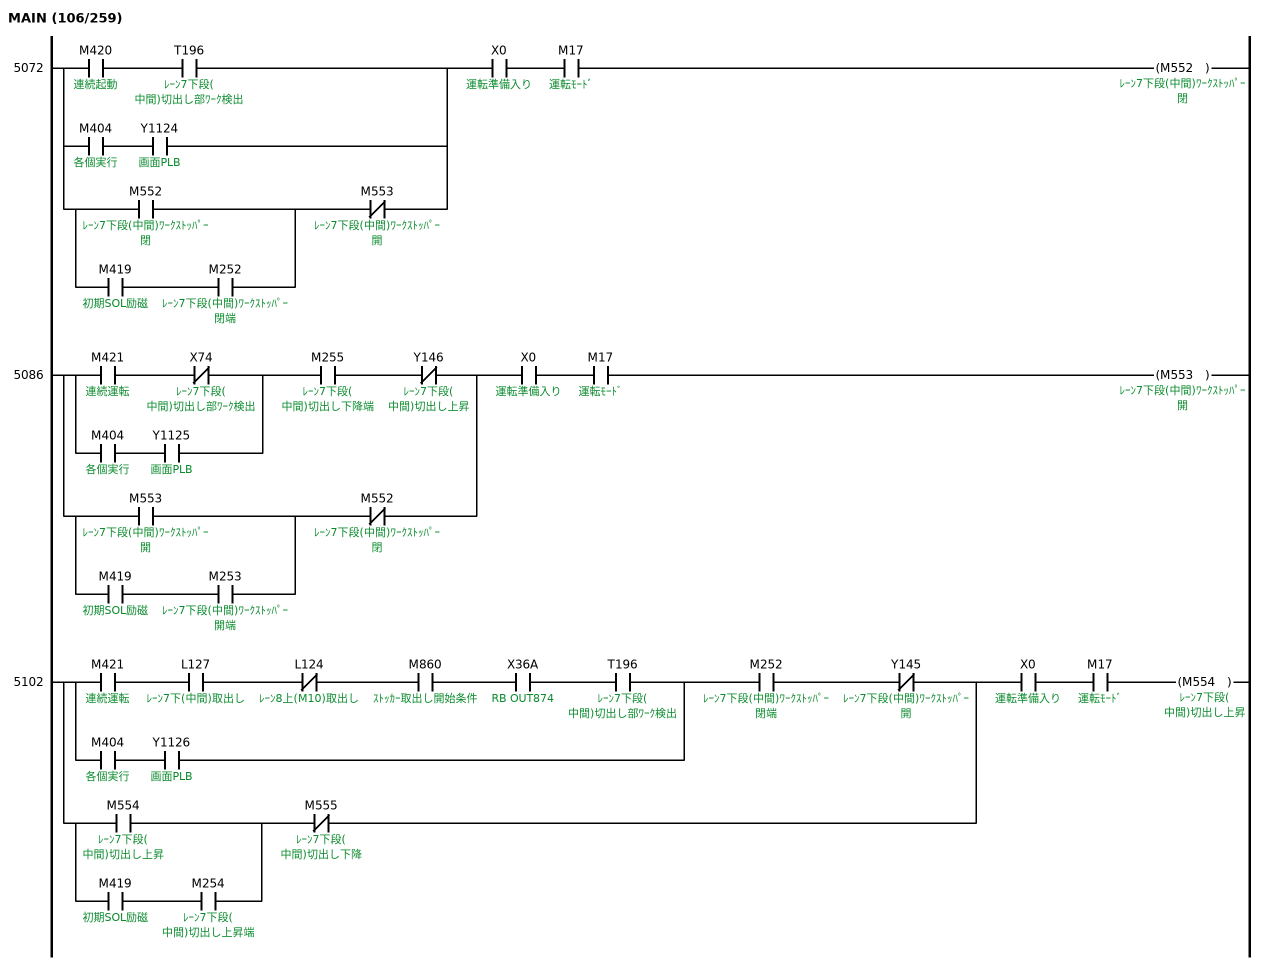
5072  LD      M420  ; 連続起動
      AND     T196  ; ﾚｰﾝ7下段(中間)切出し部ﾜｰｸ検出
      LD      M404  ; 各個実行
      AND     Y1124  ; 画面PLB
      ORB
      LD      M552  ; ﾚｰﾝ7下段(中間)ﾜｰｸｽﾄｯﾊﾟｰ閉
      LD      M419  ; 初期SOL励磁
      AND     M252  ; ﾚｰﾝ7下段(中間)ﾜｰｸｽﾄｯﾊﾟｰ閉端
      ORB
      ANI     M553  ; ﾚｰﾝ7下段(中間)ﾜｰｸｽﾄｯﾊﾟｰ開
      ORB
      AND     X0  ; 運転準備入り
      AND     M17  ; 運転ﾓｰﾄﾞ
      OUT     M552  ; ﾚｰﾝ7下段(中間)ﾜｰｸｽﾄｯﾊﾟｰ閉
5086  LD      M421  ; 連続運転
      ANI     X74  ; ﾚｰﾝ7下段(中間)切出し部ﾜｰｸ検出
      LD      M404  ; 各個実行
      AND     Y1125  ; 画面PLB
      ORB
      AND     M255  ; ﾚｰﾝ7下段(中間)切出し下降端
      ANI     Y146  ; ﾚｰﾝ7下段(中間)切出し上昇
      LD      M553  ; ﾚｰﾝ7下段(中間)ﾜｰｸｽﾄｯﾊﾟｰ開
      LD      M419  ; 初期SOL励磁
      AND     M253  ; ﾚｰﾝ7下段(中間)ﾜｰｸｽﾄｯﾊﾟｰ開端
      ORB
      ANI     M552  ; ﾚｰﾝ7下段(中間)ﾜｰｸｽﾄｯﾊﾟｰ閉
      ORB
      AND     X0  ; 運転準備入り
      AND     M17  ; 運転ﾓｰﾄﾞ
      OUT     M553  ; ﾚｰﾝ7下段(中間)ﾜｰｸｽﾄｯﾊﾟｰ開
5102  LD      M421  ; 連続運転
      AND     L127  ; ﾚｰﾝ7下(中間)取出し
      ANI     L124  ; ﾚｰﾝ8上(M10)取出し
      AND     M860  ; ｽﾄｯｶｰ取出し開始条件
      AND     X36A  ; RB OUT874
      AND     T196  ; ﾚｰﾝ7下段(中間)切出し部ﾜｰｸ検出
      LD      M404  ; 各個実行
      AND     Y1126  ; 画面PLB
      ORB
      AND     M252  ; ﾚｰﾝ7下段(中間)ﾜｰｸｽﾄｯﾊﾟｰ閉端
      ANI     Y145  ; ﾚｰﾝ7下段(中間)ﾜｰｸｽﾄｯﾊﾟｰ開
      LD      M554  ; ﾚｰﾝ7下段(中間)切出し上昇
      LD      M419  ; 初期SOL励磁
      AND     M254  ; ﾚｰﾝ7下段(中間)切出し上昇端
      ORB
      ANI     M555  ; ﾚｰﾝ7下段(中間)切出し下降
      ORB
      AND     X0  ; 運転準備入り
      AND     M17  ; 運転ﾓｰﾄﾞ
      OUT     M554  ; ﾚｰﾝ7下段(中間)切出し上昇
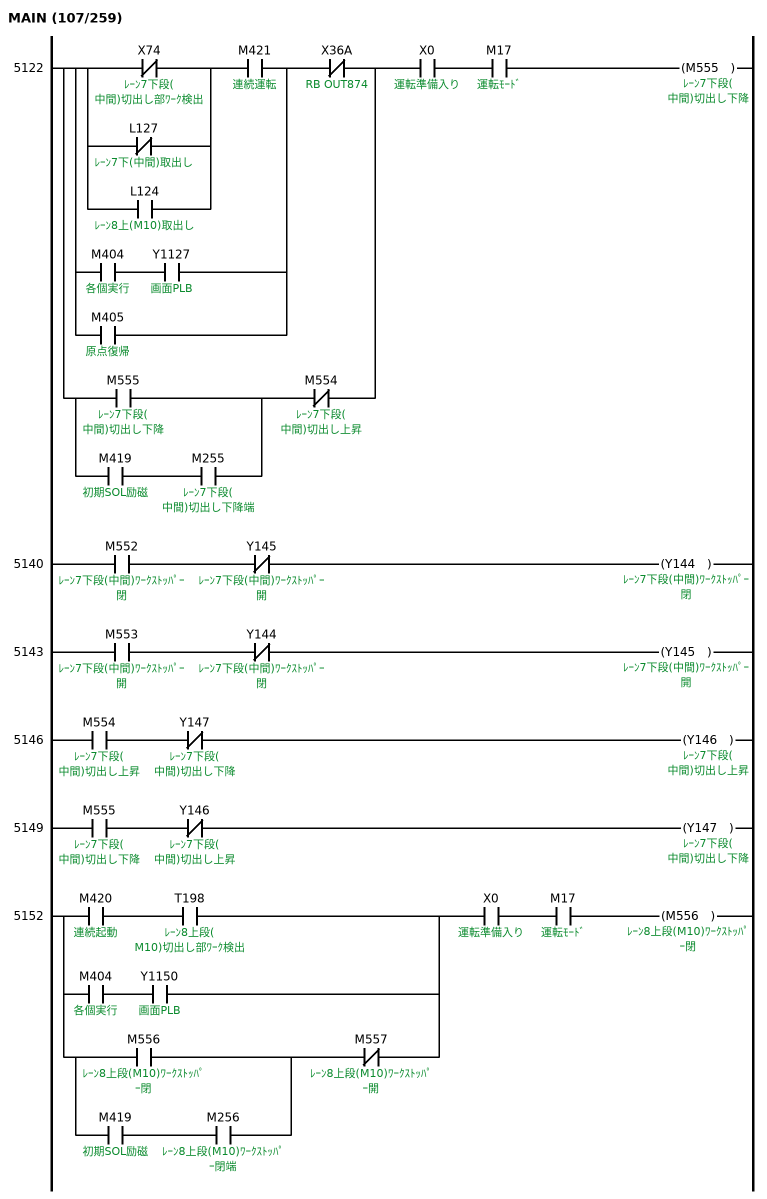
5122  LDI     X74  ; ﾚｰﾝ7下段(中間)切出し部ﾜｰｸ検出
      ORI     L127  ; ﾚｰﾝ7下(中間)取出し
      OR      L124  ; ﾚｰﾝ8上(M10)取出し
      AND     M421  ; 連続運転
      LD      M404  ; 各個実行
      AND     Y1127  ; 画面PLB
      ORB
      OR      M405  ; 原点復帰
      ANI     X36A  ; RB OUT874
      LD      M555  ; ﾚｰﾝ7下段(中間)切出し下降
      LD      M419  ; 初期SOL励磁
      AND     M255  ; ﾚｰﾝ7下段(中間)切出し下降端
      ORB
      ANI     M554  ; ﾚｰﾝ7下段(中間)切出し上昇
      ORB
      AND     X0  ; 運転準備入り
      AND     M17  ; 運転ﾓｰﾄﾞ
      OUT     M555  ; ﾚｰﾝ7下段(中間)切出し下降
5140  LD      M552  ; ﾚｰﾝ7下段(中間)ﾜｰｸｽﾄｯﾊﾟｰ閉
      ANI     Y145  ; ﾚｰﾝ7下段(中間)ﾜｰｸｽﾄｯﾊﾟｰ開
      OUT     Y144  ; ﾚｰﾝ7下段(中間)ﾜｰｸｽﾄｯﾊﾟｰ閉
5143  LD      M553  ; ﾚｰﾝ7下段(中間)ﾜｰｸｽﾄｯﾊﾟｰ開
      ANI     Y144  ; ﾚｰﾝ7下段(中間)ﾜｰｸｽﾄｯﾊﾟｰ閉
      OUT     Y145  ; ﾚｰﾝ7下段(中間)ﾜｰｸｽﾄｯﾊﾟｰ開
5146  LD      M554  ; ﾚｰﾝ7下段(中間)切出し上昇
      ANI     Y147  ; ﾚｰﾝ7下段(中間)切出し下降
      OUT     Y146  ; ﾚｰﾝ7下段(中間)切出し上昇
5149  LD      M555  ; ﾚｰﾝ7下段(中間)切出し下降
      ANI     Y146  ; ﾚｰﾝ7下段(中間)切出し上昇
      OUT     Y147  ; ﾚｰﾝ7下段(中間)切出し下降
5152  LD      M420  ; 連続起動
      AND     T198  ; ﾚｰﾝ8上段(M10)切出し部ﾜｰｸ検出
      LD      M404  ; 各個実行
      AND     Y1150  ; 画面PLB
      ORB
      LD      M556  ; ﾚｰﾝ8上段(M10)ﾜｰｸｽﾄｯﾊﾟｰ閉
      LD      M419  ; 初期SOL励磁
      AND     M256  ; ﾚｰﾝ8上段(M10)ﾜｰｸｽﾄｯﾊﾟｰ閉端
      ORB
      ANI     M557  ; ﾚｰﾝ8上段(M10)ﾜｰｸｽﾄｯﾊﾟｰ開
      ORB
      AND     X0  ; 運転準備入り
      AND     M17  ; 運転ﾓｰﾄﾞ
      OUT     M556  ; ﾚｰﾝ8上段(M10)ﾜｰｸｽﾄｯﾊﾟｰ閉
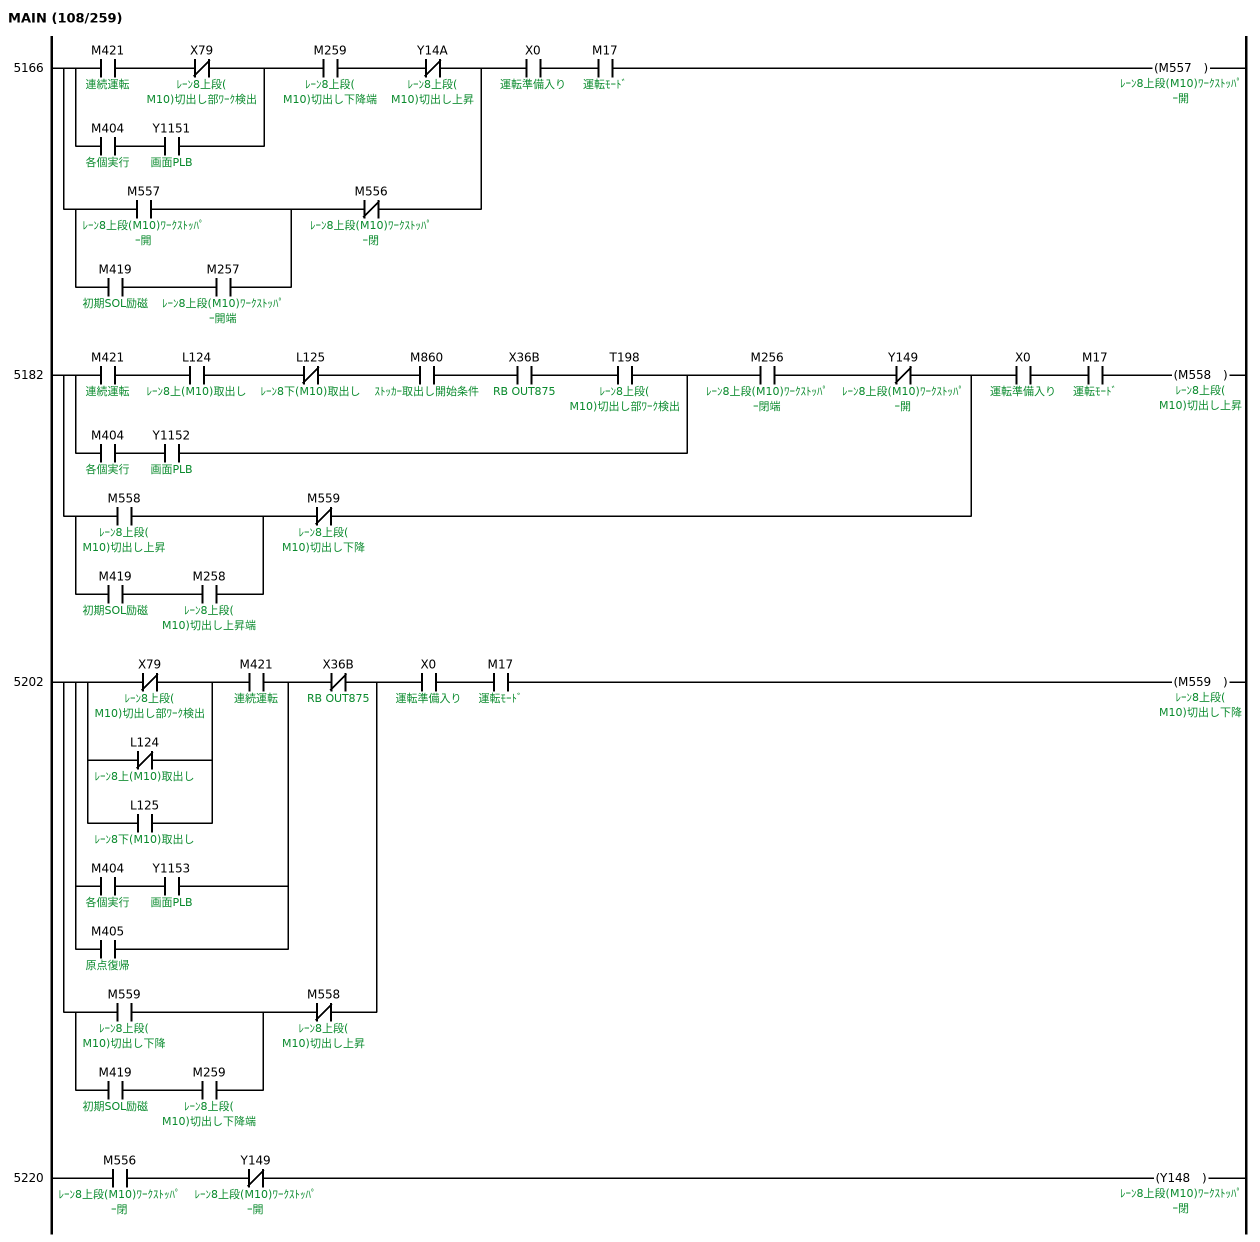
5166  LD      M421  ; 連続運転
      ANI     X79  ; ﾚｰﾝ8上段(M10)切出し部ﾜｰｸ検出
      LD      M404  ; 各個実行
      AND     Y1151  ; 画面PLB
      ORB
      AND     M259  ; ﾚｰﾝ8上段(M10)切出し下降端
      ANI     Y14A  ; ﾚｰﾝ8上段(M10)切出し上昇
      LD      M557  ; ﾚｰﾝ8上段(M10)ﾜｰｸｽﾄｯﾊﾟｰ開
      LD      M419  ; 初期SOL励磁
      AND     M257  ; ﾚｰﾝ8上段(M10)ﾜｰｸｽﾄｯﾊﾟｰ開端
      ORB
      ANI     M556  ; ﾚｰﾝ8上段(M10)ﾜｰｸｽﾄｯﾊﾟｰ閉
      ORB
      AND     X0  ; 運転準備入り
      AND     M17  ; 運転ﾓｰﾄﾞ
      OUT     M557  ; ﾚｰﾝ8上段(M10)ﾜｰｸｽﾄｯﾊﾟｰ開
5182  LD      M421  ; 連続運転
      AND     L124  ; ﾚｰﾝ8上(M10)取出し
      ANI     L125  ; ﾚｰﾝ8下(M10)取出し
      AND     M860  ; ｽﾄｯｶｰ取出し開始条件
      AND     X36B  ; RB OUT875
      AND     T198  ; ﾚｰﾝ8上段(M10)切出し部ﾜｰｸ検出
      LD      M404  ; 各個実行
      AND     Y1152  ; 画面PLB
      ORB
      AND     M256  ; ﾚｰﾝ8上段(M10)ﾜｰｸｽﾄｯﾊﾟｰ閉端
      ANI     Y149  ; ﾚｰﾝ8上段(M10)ﾜｰｸｽﾄｯﾊﾟｰ開
      LD      M558  ; ﾚｰﾝ8上段(M10)切出し上昇
      LD      M419  ; 初期SOL励磁
      AND     M258  ; ﾚｰﾝ8上段(M10)切出し上昇端
      ORB
      ANI     M559  ; ﾚｰﾝ8上段(M10)切出し下降
      ORB
      AND     X0  ; 運転準備入り
      AND     M17  ; 運転ﾓｰﾄﾞ
      OUT     M558  ; ﾚｰﾝ8上段(M10)切出し上昇
5202  LDI     X79  ; ﾚｰﾝ8上段(M10)切出し部ﾜｰｸ検出
      ORI     L124  ; ﾚｰﾝ8上(M10)取出し
      OR      L125  ; ﾚｰﾝ8下(M10)取出し
      AND     M421  ; 連続運転
      LD      M404  ; 各個実行
      AND     Y1153  ; 画面PLB
      ORB
      OR      M405  ; 原点復帰
      ANI     X36B  ; RB OUT875
      LD      M559  ; ﾚｰﾝ8上段(M10)切出し下降
      LD      M419  ; 初期SOL励磁
      AND     M259  ; ﾚｰﾝ8上段(M10)切出し下降端
      ORB
      ANI     M558  ; ﾚｰﾝ8上段(M10)切出し上昇
      ORB
      AND     X0  ; 運転準備入り
      AND     M17  ; 運転ﾓｰﾄﾞ
      OUT     M559  ; ﾚｰﾝ8上段(M10)切出し下降
5220  LD      M556  ; ﾚｰﾝ8上段(M10)ﾜｰｸｽﾄｯﾊﾟｰ閉
      ANI     Y149  ; ﾚｰﾝ8上段(M10)ﾜｰｸｽﾄｯﾊﾟｰ開
      OUT     Y148  ; ﾚｰﾝ8上段(M10)ﾜｰｸｽﾄｯﾊﾟｰ閉
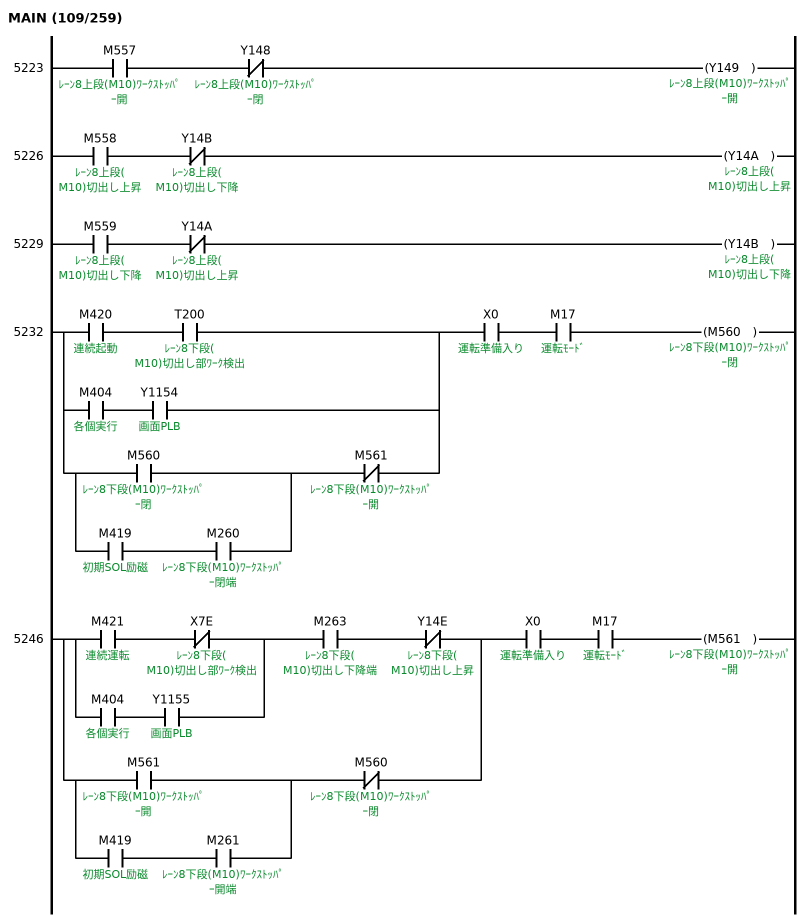
5223  LD      M557  ; ﾚｰﾝ8上段(M10)ﾜｰｸｽﾄｯﾊﾟｰ開
      ANI     Y148  ; ﾚｰﾝ8上段(M10)ﾜｰｸｽﾄｯﾊﾟｰ閉
      OUT     Y149  ; ﾚｰﾝ8上段(M10)ﾜｰｸｽﾄｯﾊﾟｰ開
5226  LD      M558  ; ﾚｰﾝ8上段(M10)切出し上昇
      ANI     Y14B  ; ﾚｰﾝ8上段(M10)切出し下降
      OUT     Y14A  ; ﾚｰﾝ8上段(M10)切出し上昇
5229  LD      M559  ; ﾚｰﾝ8上段(M10)切出し下降
      ANI     Y14A  ; ﾚｰﾝ8上段(M10)切出し上昇
      OUT     Y14B  ; ﾚｰﾝ8上段(M10)切出し下降
5232  LD      M420  ; 連続起動
      AND     T200  ; ﾚｰﾝ8下段(M10)切出し部ﾜｰｸ検出
      LD      M404  ; 各個実行
      AND     Y1154  ; 画面PLB
      ORB
      LD      M560  ; ﾚｰﾝ8下段(M10)ﾜｰｸｽﾄｯﾊﾟｰ閉
      LD      M419  ; 初期SOL励磁
      AND     M260  ; ﾚｰﾝ8下段(M10)ﾜｰｸｽﾄｯﾊﾟｰ閉端
      ORB
      ANI     M561  ; ﾚｰﾝ8下段(M10)ﾜｰｸｽﾄｯﾊﾟｰ開
      ORB
      AND     X0  ; 運転準備入り
      AND     M17  ; 運転ﾓｰﾄﾞ
      OUT     M560  ; ﾚｰﾝ8下段(M10)ﾜｰｸｽﾄｯﾊﾟｰ閉
5246  LD      M421  ; 連続運転
      ANI     X7E  ; ﾚｰﾝ8下段(M10)切出し部ﾜｰｸ検出
      LD      M404  ; 各個実行
      AND     Y1155  ; 画面PLB
      ORB
      AND     M263  ; ﾚｰﾝ8下段(M10)切出し下降端
      ANI     Y14E  ; ﾚｰﾝ8下段(M10)切出し上昇
      LD      M561  ; ﾚｰﾝ8下段(M10)ﾜｰｸｽﾄｯﾊﾟｰ開
      LD      M419  ; 初期SOL励磁
      AND     M261  ; ﾚｰﾝ8下段(M10)ﾜｰｸｽﾄｯﾊﾟｰ開端
      ORB
      ANI     M560  ; ﾚｰﾝ8下段(M10)ﾜｰｸｽﾄｯﾊﾟｰ閉
      ORB
      AND     X0  ; 運転準備入り
      AND     M17  ; 運転ﾓｰﾄﾞ
      OUT     M561  ; ﾚｰﾝ8下段(M10)ﾜｰｸｽﾄｯﾊﾟｰ開
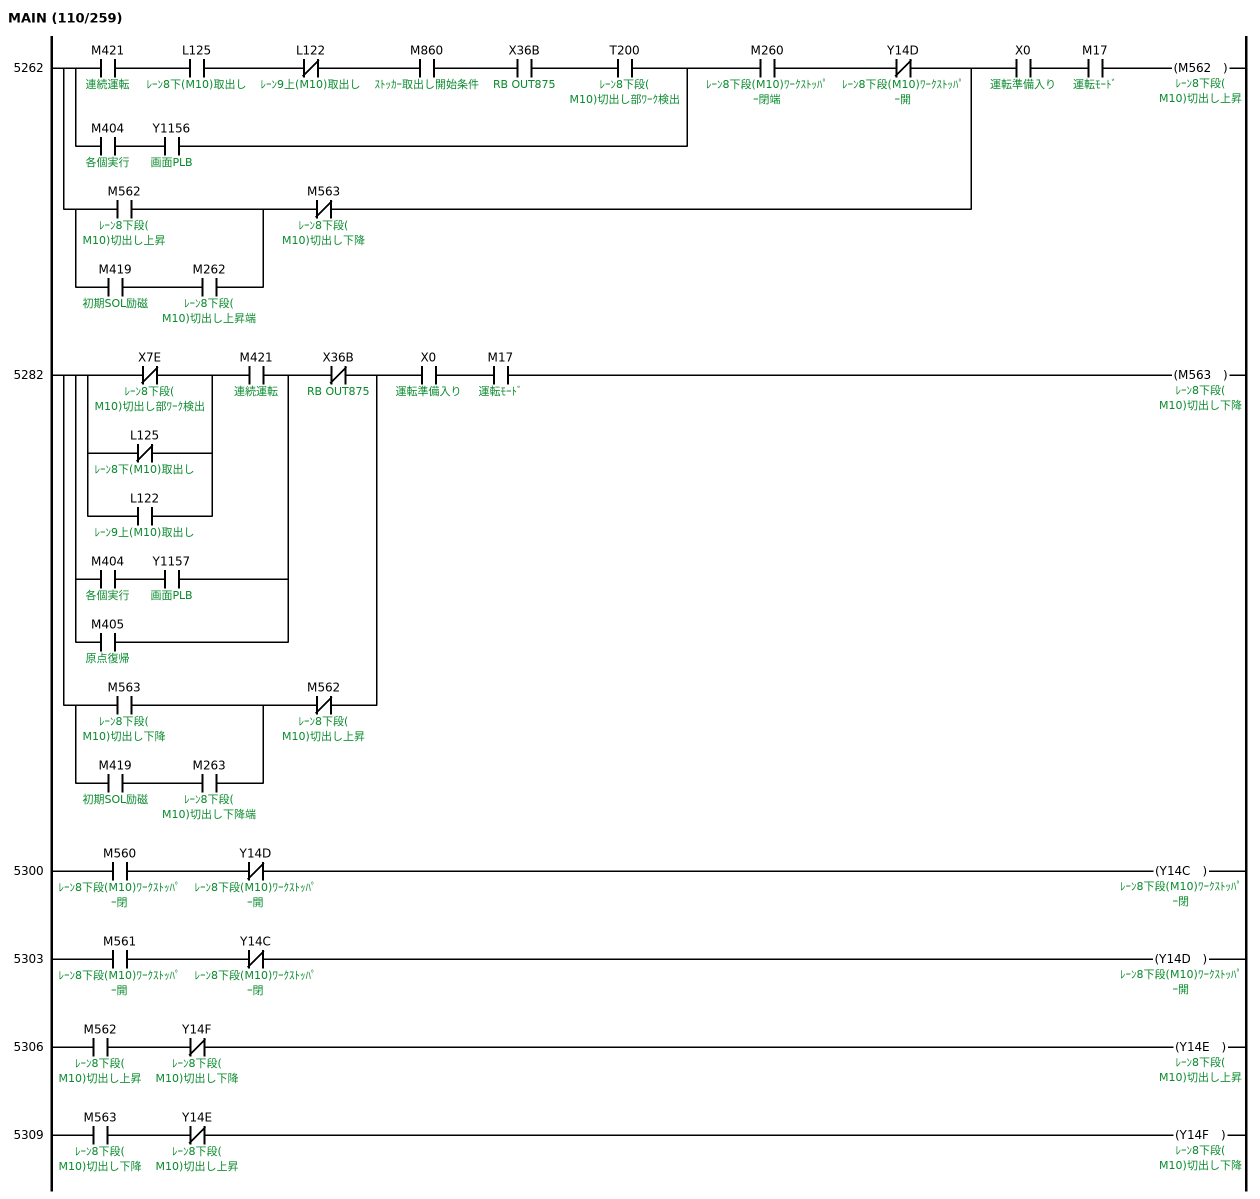
5262  LD      M421  ; 連続運転
      AND     L125  ; ﾚｰﾝ8下(M10)取出し
      ANI     L122  ; ﾚｰﾝ9上(M10)取出し
      AND     M860  ; ｽﾄｯｶｰ取出し開始条件
      AND     X36B  ; RB OUT875
      AND     T200  ; ﾚｰﾝ8下段(M10)切出し部ﾜｰｸ検出
      LD      M404  ; 各個実行
      AND     Y1156  ; 画面PLB
      ORB
      AND     M260  ; ﾚｰﾝ8下段(M10)ﾜｰｸｽﾄｯﾊﾟｰ閉端
      ANI     Y14D  ; ﾚｰﾝ8下段(M10)ﾜｰｸｽﾄｯﾊﾟｰ開
      LD      M562  ; ﾚｰﾝ8下段(M10)切出し上昇
      LD      M419  ; 初期SOL励磁
      AND     M262  ; ﾚｰﾝ8下段(M10)切出し上昇端
      ORB
      ANI     M563  ; ﾚｰﾝ8下段(M10)切出し下降
      ORB
      AND     X0  ; 運転準備入り
      AND     M17  ; 運転ﾓｰﾄﾞ
      OUT     M562  ; ﾚｰﾝ8下段(M10)切出し上昇
5282  LDI     X7E  ; ﾚｰﾝ8下段(M10)切出し部ﾜｰｸ検出
      ORI     L125  ; ﾚｰﾝ8下(M10)取出し
      OR      L122  ; ﾚｰﾝ9上(M10)取出し
      AND     M421  ; 連続運転
      LD      M404  ; 各個実行
      AND     Y1157  ; 画面PLB
      ORB
      OR      M405  ; 原点復帰
      ANI     X36B  ; RB OUT875
      LD      M563  ; ﾚｰﾝ8下段(M10)切出し下降
      LD      M419  ; 初期SOL励磁
      AND     M263  ; ﾚｰﾝ8下段(M10)切出し下降端
      ORB
      ANI     M562  ; ﾚｰﾝ8下段(M10)切出し上昇
      ORB
      AND     X0  ; 運転準備入り
      AND     M17  ; 運転ﾓｰﾄﾞ
      OUT     M563  ; ﾚｰﾝ8下段(M10)切出し下降
5300  LD      M560  ; ﾚｰﾝ8下段(M10)ﾜｰｸｽﾄｯﾊﾟｰ閉
      ANI     Y14D  ; ﾚｰﾝ8下段(M10)ﾜｰｸｽﾄｯﾊﾟｰ開
      OUT     Y14C  ; ﾚｰﾝ8下段(M10)ﾜｰｸｽﾄｯﾊﾟｰ閉
5303  LD      M561  ; ﾚｰﾝ8下段(M10)ﾜｰｸｽﾄｯﾊﾟｰ開
      ANI     Y14C  ; ﾚｰﾝ8下段(M10)ﾜｰｸｽﾄｯﾊﾟｰ閉
      OUT     Y14D  ; ﾚｰﾝ8下段(M10)ﾜｰｸｽﾄｯﾊﾟｰ開
5306  LD      M562  ; ﾚｰﾝ8下段(M10)切出し上昇
      ANI     Y14F  ; ﾚｰﾝ8下段(M10)切出し下降
      OUT     Y14E  ; ﾚｰﾝ8下段(M10)切出し上昇
5309  LD      M563  ; ﾚｰﾝ8下段(M10)切出し下降
      ANI     Y14E  ; ﾚｰﾝ8下段(M10)切出し上昇
      OUT     Y14F  ; ﾚｰﾝ8下段(M10)切出し下降
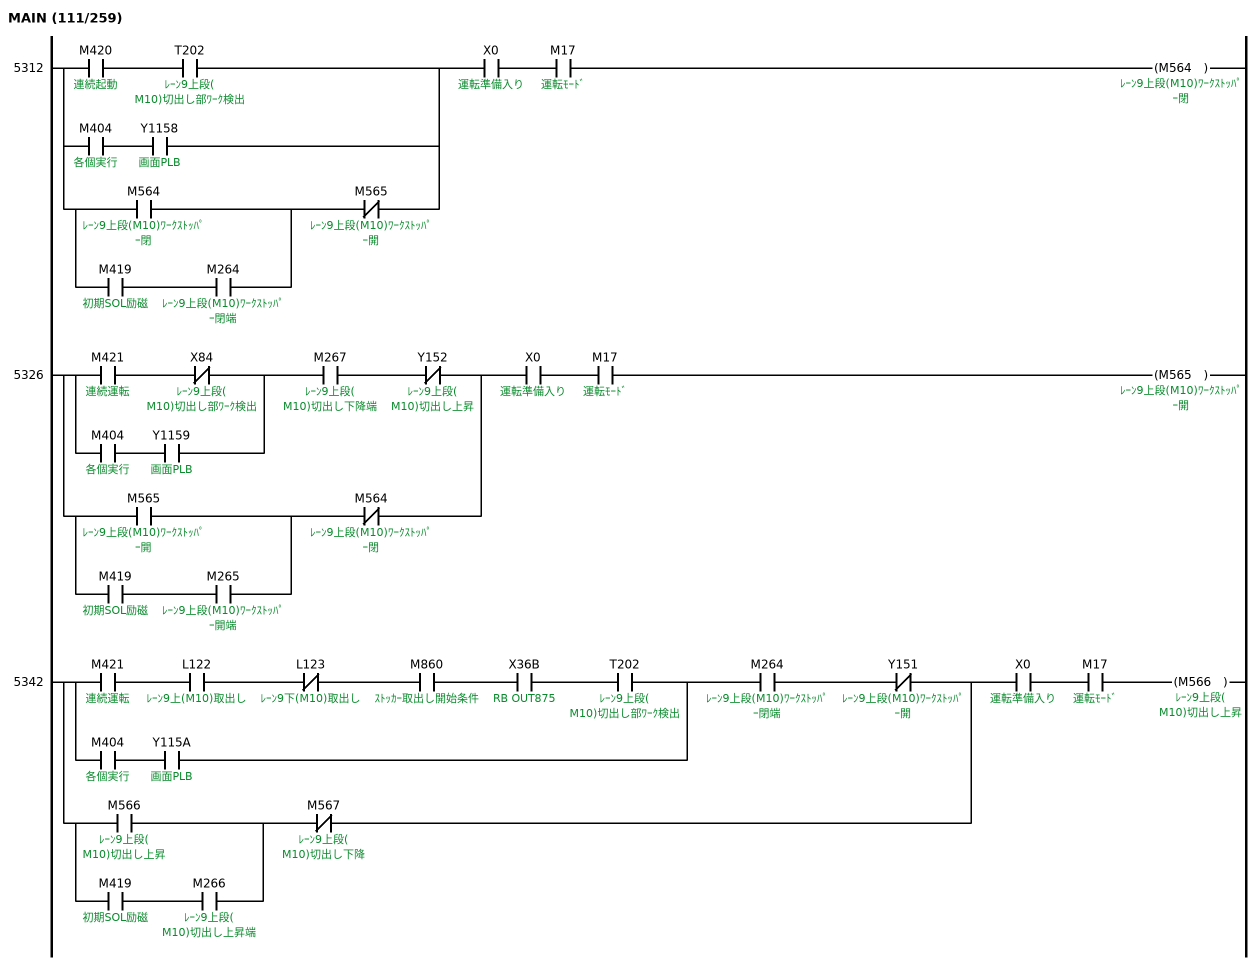
5312  LD      M420  ; 連続起動
      AND     T202  ; ﾚｰﾝ9上段(M10)切出し部ﾜｰｸ検出
      LD      M404  ; 各個実行
      AND     Y1158  ; 画面PLB
      ORB
      LD      M564  ; ﾚｰﾝ9上段(M10)ﾜｰｸｽﾄｯﾊﾟｰ閉
      LD      M419  ; 初期SOL励磁
      AND     M264  ; ﾚｰﾝ9上段(M10)ﾜｰｸｽﾄｯﾊﾟｰ閉端
      ORB
      ANI     M565  ; ﾚｰﾝ9上段(M10)ﾜｰｸｽﾄｯﾊﾟｰ開
      ORB
      AND     X0  ; 運転準備入り
      AND     M17  ; 運転ﾓｰﾄﾞ
      OUT     M564  ; ﾚｰﾝ9上段(M10)ﾜｰｸｽﾄｯﾊﾟｰ閉
5326  LD      M421  ; 連続運転
      ANI     X84  ; ﾚｰﾝ9上段(M10)切出し部ﾜｰｸ検出
      LD      M404  ; 各個実行
      AND     Y1159  ; 画面PLB
      ORB
      AND     M267  ; ﾚｰﾝ9上段(M10)切出し下降端
      ANI     Y152  ; ﾚｰﾝ9上段(M10)切出し上昇
      LD      M565  ; ﾚｰﾝ9上段(M10)ﾜｰｸｽﾄｯﾊﾟｰ開
      LD      M419  ; 初期SOL励磁
      AND     M265  ; ﾚｰﾝ9上段(M10)ﾜｰｸｽﾄｯﾊﾟｰ開端
      ORB
      ANI     M564  ; ﾚｰﾝ9上段(M10)ﾜｰｸｽﾄｯﾊﾟｰ閉
      ORB
      AND     X0  ; 運転準備入り
      AND     M17  ; 運転ﾓｰﾄﾞ
      OUT     M565  ; ﾚｰﾝ9上段(M10)ﾜｰｸｽﾄｯﾊﾟｰ開
5342  LD      M421  ; 連続運転
      AND     L122  ; ﾚｰﾝ9上(M10)取出し
      ANI     L123  ; ﾚｰﾝ9下(M10)取出し
      AND     M860  ; ｽﾄｯｶｰ取出し開始条件
      AND     X36B  ; RB OUT875
      AND     T202  ; ﾚｰﾝ9上段(M10)切出し部ﾜｰｸ検出
      LD      M404  ; 各個実行
      AND     Y115A  ; 画面PLB
      ORB
      AND     M264  ; ﾚｰﾝ9上段(M10)ﾜｰｸｽﾄｯﾊﾟｰ閉端
      ANI     Y151  ; ﾚｰﾝ9上段(M10)ﾜｰｸｽﾄｯﾊﾟｰ開
      LD      M566  ; ﾚｰﾝ9上段(M10)切出し上昇
      LD      M419  ; 初期SOL励磁
      AND     M266  ; ﾚｰﾝ9上段(M10)切出し上昇端
      ORB
      ANI     M567  ; ﾚｰﾝ9上段(M10)切出し下降
      ORB
      AND     X0  ; 運転準備入り
      AND     M17  ; 運転ﾓｰﾄﾞ
      OUT     M566  ; ﾚｰﾝ9上段(M10)切出し上昇
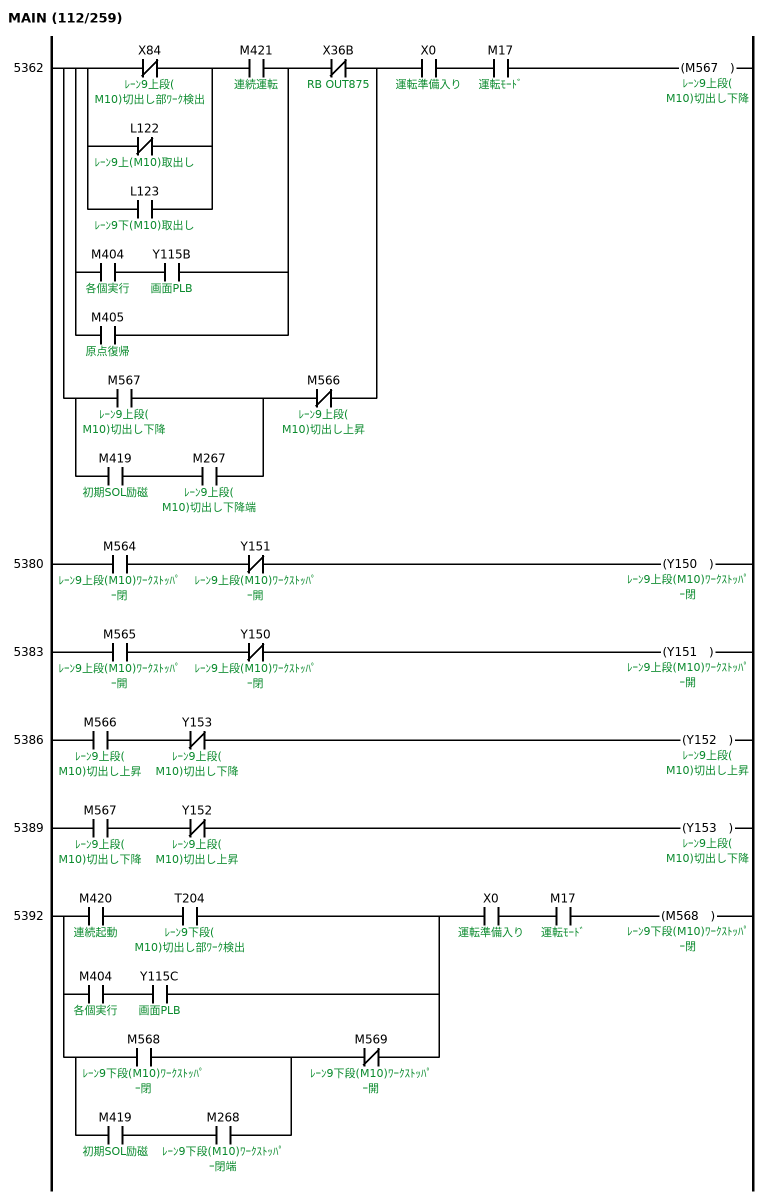
5362  LDI     X84  ; ﾚｰﾝ9上段(M10)切出し部ﾜｰｸ検出
      ORI     L122  ; ﾚｰﾝ9上(M10)取出し
      OR      L123  ; ﾚｰﾝ9下(M10)取出し
      AND     M421  ; 連続運転
      LD      M404  ; 各個実行
      AND     Y115B  ; 画面PLB
      ORB
      OR      M405  ; 原点復帰
      ANI     X36B  ; RB OUT875
      LD      M567  ; ﾚｰﾝ9上段(M10)切出し下降
      LD      M419  ; 初期SOL励磁
      AND     M267  ; ﾚｰﾝ9上段(M10)切出し下降端
      ORB
      ANI     M566  ; ﾚｰﾝ9上段(M10)切出し上昇
      ORB
      AND     X0  ; 運転準備入り
      AND     M17  ; 運転ﾓｰﾄﾞ
      OUT     M567  ; ﾚｰﾝ9上段(M10)切出し下降
5380  LD      M564  ; ﾚｰﾝ9上段(M10)ﾜｰｸｽﾄｯﾊﾟｰ閉
      ANI     Y151  ; ﾚｰﾝ9上段(M10)ﾜｰｸｽﾄｯﾊﾟｰ開
      OUT     Y150  ; ﾚｰﾝ9上段(M10)ﾜｰｸｽﾄｯﾊﾟｰ閉
5383  LD      M565  ; ﾚｰﾝ9上段(M10)ﾜｰｸｽﾄｯﾊﾟｰ開
      ANI     Y150  ; ﾚｰﾝ9上段(M10)ﾜｰｸｽﾄｯﾊﾟｰ閉
      OUT     Y151  ; ﾚｰﾝ9上段(M10)ﾜｰｸｽﾄｯﾊﾟｰ開
5386  LD      M566  ; ﾚｰﾝ9上段(M10)切出し上昇
      ANI     Y153  ; ﾚｰﾝ9上段(M10)切出し下降
      OUT     Y152  ; ﾚｰﾝ9上段(M10)切出し上昇
5389  LD      M567  ; ﾚｰﾝ9上段(M10)切出し下降
      ANI     Y152  ; ﾚｰﾝ9上段(M10)切出し上昇
      OUT     Y153  ; ﾚｰﾝ9上段(M10)切出し下降
5392  LD      M420  ; 連続起動
      AND     T204  ; ﾚｰﾝ9下段(M10)切出し部ﾜｰｸ検出
      LD      M404  ; 各個実行
      AND     Y115C  ; 画面PLB
      ORB
      LD      M568  ; ﾚｰﾝ9下段(M10)ﾜｰｸｽﾄｯﾊﾟｰ閉
      LD      M419  ; 初期SOL励磁
      AND     M268  ; ﾚｰﾝ9下段(M10)ﾜｰｸｽﾄｯﾊﾟｰ閉端
      ORB
      ANI     M569  ; ﾚｰﾝ9下段(M10)ﾜｰｸｽﾄｯﾊﾟｰ開
      ORB
      AND     X0  ; 運転準備入り
      AND     M17  ; 運転ﾓｰﾄﾞ
      OUT     M568  ; ﾚｰﾝ9下段(M10)ﾜｰｸｽﾄｯﾊﾟｰ閉
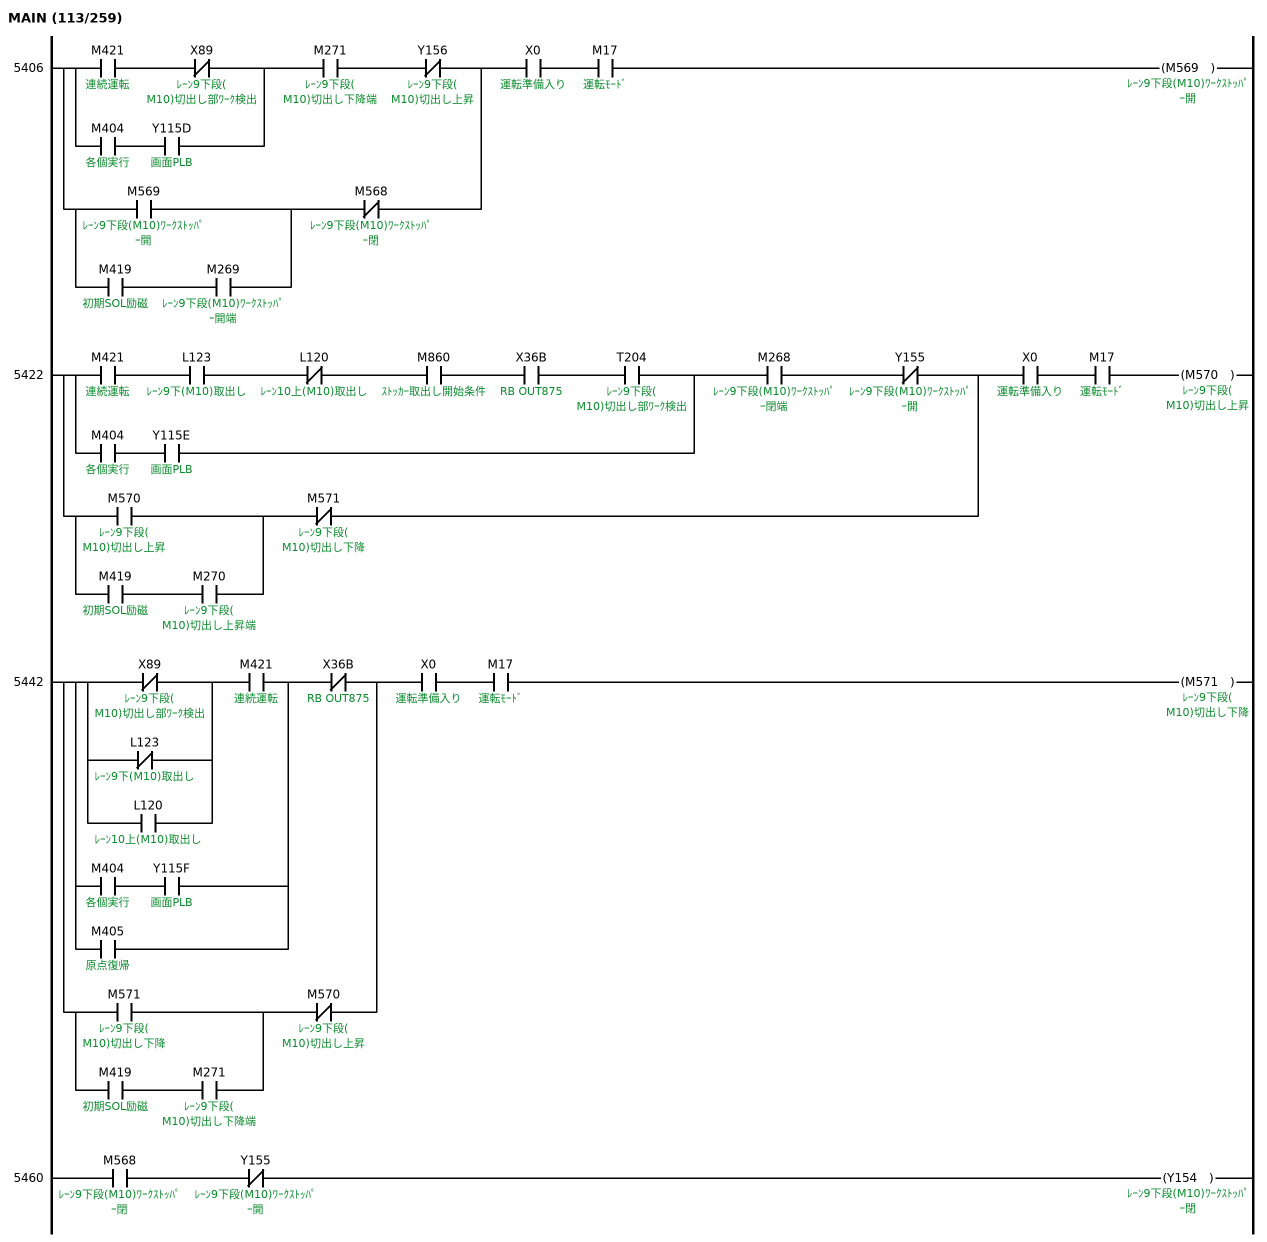
5406  LD      M421  ; 連続運転
      ANI     X89  ; ﾚｰﾝ9下段(M10)切出し部ﾜｰｸ検出
      LD      M404  ; 各個実行
      AND     Y115D  ; 画面PLB
      ORB
      AND     M271  ; ﾚｰﾝ9下段(M10)切出し下降端
      ANI     Y156  ; ﾚｰﾝ9下段(M10)切出し上昇
      LD      M569  ; ﾚｰﾝ9下段(M10)ﾜｰｸｽﾄｯﾊﾟｰ開
      LD      M419  ; 初期SOL励磁
      AND     M269  ; ﾚｰﾝ9下段(M10)ﾜｰｸｽﾄｯﾊﾟｰ開端
      ORB
      ANI     M568  ; ﾚｰﾝ9下段(M10)ﾜｰｸｽﾄｯﾊﾟｰ閉
      ORB
      AND     X0  ; 運転準備入り
      AND     M17  ; 運転ﾓｰﾄﾞ
      OUT     M569  ; ﾚｰﾝ9下段(M10)ﾜｰｸｽﾄｯﾊﾟｰ開
5422  LD      M421  ; 連続運転
      AND     L123  ; ﾚｰﾝ9下(M10)取出し
      ANI     L120  ; ﾚｰﾝ10上(M10)取出し
      AND     M860  ; ｽﾄｯｶｰ取出し開始条件
      AND     X36B  ; RB OUT875
      AND     T204  ; ﾚｰﾝ9下段(M10)切出し部ﾜｰｸ検出
      LD      M404  ; 各個実行
      AND     Y115E  ; 画面PLB
      ORB
      AND     M268  ; ﾚｰﾝ9下段(M10)ﾜｰｸｽﾄｯﾊﾟｰ閉端
      ANI     Y155  ; ﾚｰﾝ9下段(M10)ﾜｰｸｽﾄｯﾊﾟｰ開
      LD      M570  ; ﾚｰﾝ9下段(M10)切出し上昇
      LD      M419  ; 初期SOL励磁
      AND     M270  ; ﾚｰﾝ9下段(M10)切出し上昇端
      ORB
      ANI     M571  ; ﾚｰﾝ9下段(M10)切出し下降
      ORB
      AND     X0  ; 運転準備入り
      AND     M17  ; 運転ﾓｰﾄﾞ
      OUT     M570  ; ﾚｰﾝ9下段(M10)切出し上昇
5442  LDI     X89  ; ﾚｰﾝ9下段(M10)切出し部ﾜｰｸ検出
      ORI     L123  ; ﾚｰﾝ9下(M10)取出し
      OR      L120  ; ﾚｰﾝ10上(M10)取出し
      AND     M421  ; 連続運転
      LD      M404  ; 各個実行
      AND     Y115F  ; 画面PLB
      ORB
      OR      M405  ; 原点復帰
      ANI     X36B  ; RB OUT875
      LD      M571  ; ﾚｰﾝ9下段(M10)切出し下降
      LD      M419  ; 初期SOL励磁
      AND     M271  ; ﾚｰﾝ9下段(M10)切出し下降端
      ORB
      ANI     M570  ; ﾚｰﾝ9下段(M10)切出し上昇
      ORB
      AND     X0  ; 運転準備入り
      AND     M17  ; 運転ﾓｰﾄﾞ
      OUT     M571  ; ﾚｰﾝ9下段(M10)切出し下降
5460  LD      M568  ; ﾚｰﾝ9下段(M10)ﾜｰｸｽﾄｯﾊﾟｰ閉
      ANI     Y155  ; ﾚｰﾝ9下段(M10)ﾜｰｸｽﾄｯﾊﾟｰ開
      OUT     Y154  ; ﾚｰﾝ9下段(M10)ﾜｰｸｽﾄｯﾊﾟｰ閉
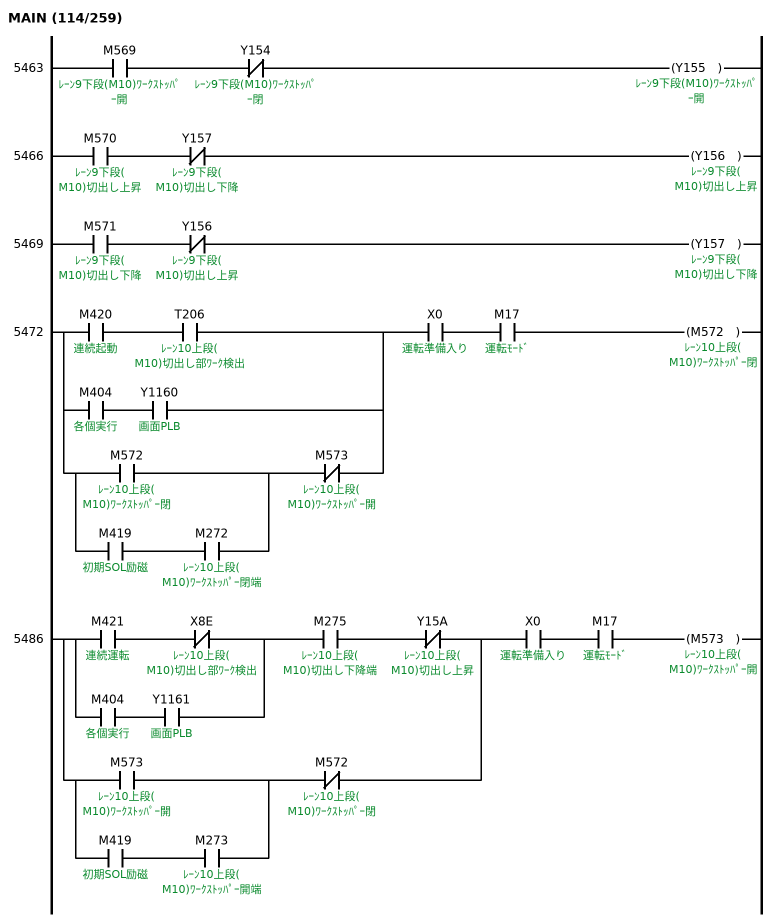
5463  LD      M569  ; ﾚｰﾝ9下段(M10)ﾜｰｸｽﾄｯﾊﾟｰ開
      ANI     Y154  ; ﾚｰﾝ9下段(M10)ﾜｰｸｽﾄｯﾊﾟｰ閉
      OUT     Y155  ; ﾚｰﾝ9下段(M10)ﾜｰｸｽﾄｯﾊﾟｰ開
5466  LD      M570  ; ﾚｰﾝ9下段(M10)切出し上昇
      ANI     Y157  ; ﾚｰﾝ9下段(M10)切出し下降
      OUT     Y156  ; ﾚｰﾝ9下段(M10)切出し上昇
5469  LD      M571  ; ﾚｰﾝ9下段(M10)切出し下降
      ANI     Y156  ; ﾚｰﾝ9下段(M10)切出し上昇
      OUT     Y157  ; ﾚｰﾝ9下段(M10)切出し下降
5472  LD      M420  ; 連続起動
      AND     T206  ; ﾚｰﾝ10上段(M10)切出し部ﾜｰｸ検出
      LD      M404  ; 各個実行
      AND     Y1160  ; 画面PLB
      ORB
      LD      M572  ; ﾚｰﾝ10上段(M10)ﾜｰｸｽﾄｯﾊﾟｰ閉
      LD      M419  ; 初期SOL励磁
      AND     M272  ; ﾚｰﾝ10上段(M10)ﾜｰｸｽﾄｯﾊﾟｰ閉端
      ORB
      ANI     M573  ; ﾚｰﾝ10上段(M10)ﾜｰｸｽﾄｯﾊﾟｰ開
      ORB
      AND     X0  ; 運転準備入り
      AND     M17  ; 運転ﾓｰﾄﾞ
      OUT     M572  ; ﾚｰﾝ10上段(M10)ﾜｰｸｽﾄｯﾊﾟｰ閉
5486  LD      M421  ; 連続運転
      ANI     X8E  ; ﾚｰﾝ10上段(M10)切出し部ﾜｰｸ検出
      LD      M404  ; 各個実行
      AND     Y1161  ; 画面PLB
      ORB
      AND     M275  ; ﾚｰﾝ10上段(M10)切出し下降端
      ANI     Y15A  ; ﾚｰﾝ10上段(M10)切出し上昇
      LD      M573  ; ﾚｰﾝ10上段(M10)ﾜｰｸｽﾄｯﾊﾟｰ開
      LD      M419  ; 初期SOL励磁
      AND     M273  ; ﾚｰﾝ10上段(M10)ﾜｰｸｽﾄｯﾊﾟｰ開端
      ORB
      ANI     M572  ; ﾚｰﾝ10上段(M10)ﾜｰｸｽﾄｯﾊﾟｰ閉
      ORB
      AND     X0  ; 運転準備入り
      AND     M17  ; 運転ﾓｰﾄﾞ
      OUT     M573  ; ﾚｰﾝ10上段(M10)ﾜｰｸｽﾄｯﾊﾟｰ開
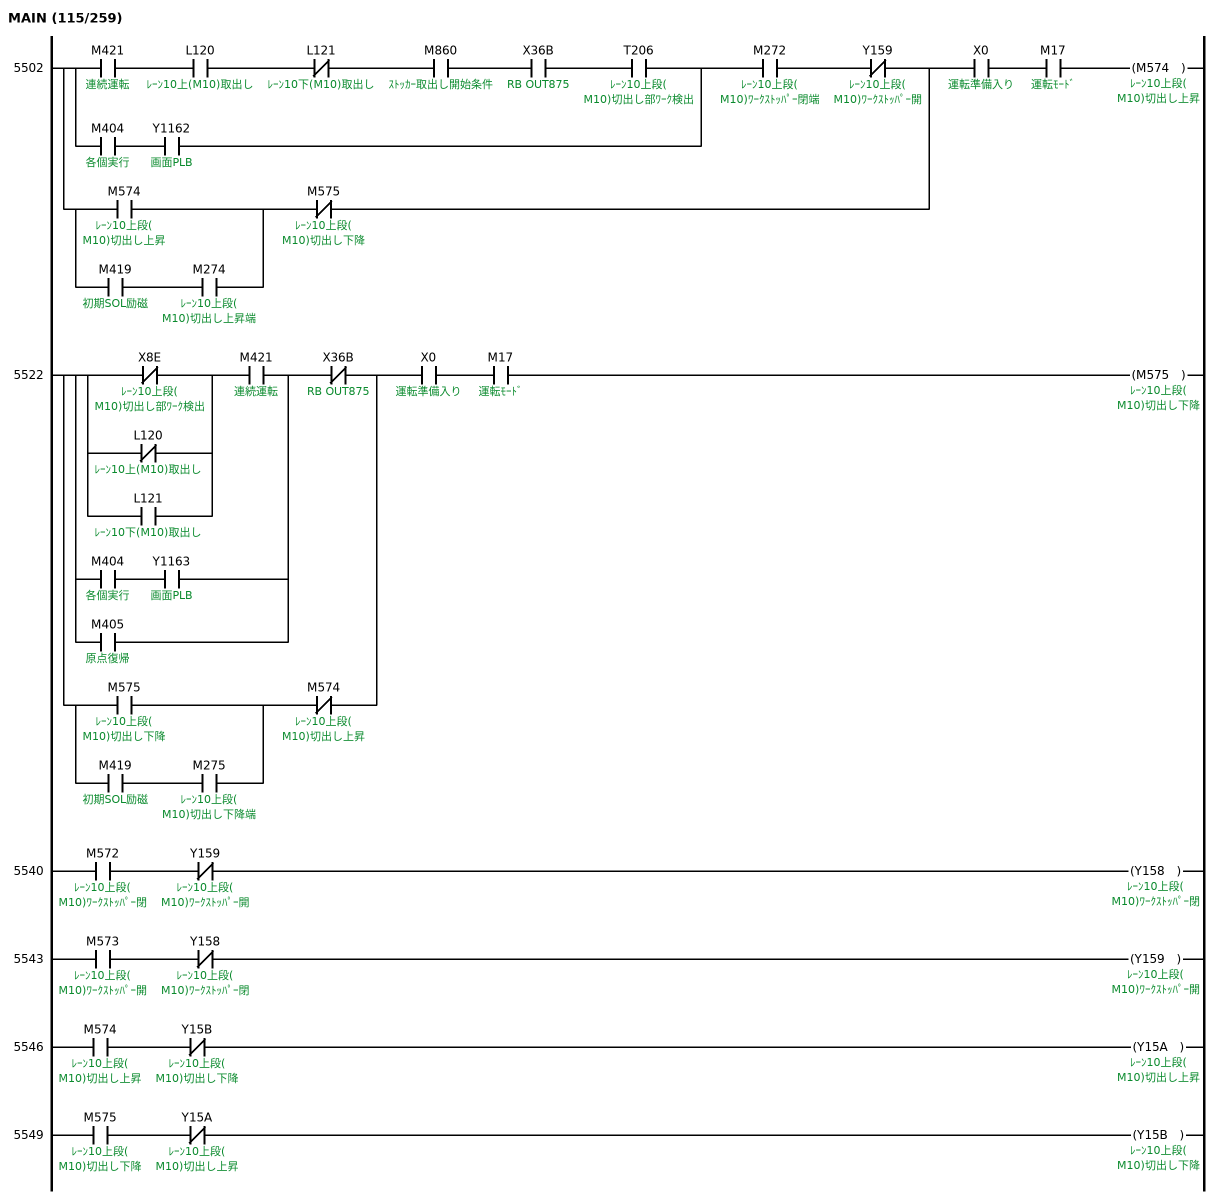
5502  LD      M421  ; 連続運転
      AND     L120  ; ﾚｰﾝ10上(M10)取出し
      ANI     L121  ; ﾚｰﾝ10下(M10)取出し
      AND     M860  ; ｽﾄｯｶｰ取出し開始条件
      AND     X36B  ; RB OUT875
      AND     T206  ; ﾚｰﾝ10上段(M10)切出し部ﾜｰｸ検出
      LD      M404  ; 各個実行
      AND     Y1162  ; 画面PLB
      ORB
      AND     M272  ; ﾚｰﾝ10上段(M10)ﾜｰｸｽﾄｯﾊﾟｰ閉端
      ANI     Y159  ; ﾚｰﾝ10上段(M10)ﾜｰｸｽﾄｯﾊﾟｰ開
      LD      M574  ; ﾚｰﾝ10上段(M10)切出し上昇
      LD      M419  ; 初期SOL励磁
      AND     M274  ; ﾚｰﾝ10上段(M10)切出し上昇端
      ORB
      ANI     M575  ; ﾚｰﾝ10上段(M10)切出し下降
      ORB
      AND     X0  ; 運転準備入り
      AND     M17  ; 運転ﾓｰﾄﾞ
      OUT     M574  ; ﾚｰﾝ10上段(M10)切出し上昇
5522  LDI     X8E  ; ﾚｰﾝ10上段(M10)切出し部ﾜｰｸ検出
      ORI     L120  ; ﾚｰﾝ10上(M10)取出し
      OR      L121  ; ﾚｰﾝ10下(M10)取出し
      AND     M421  ; 連続運転
      LD      M404  ; 各個実行
      AND     Y1163  ; 画面PLB
      ORB
      OR      M405  ; 原点復帰
      ANI     X36B  ; RB OUT875
      LD      M575  ; ﾚｰﾝ10上段(M10)切出し下降
      LD      M419  ; 初期SOL励磁
      AND     M275  ; ﾚｰﾝ10上段(M10)切出し下降端
      ORB
      ANI     M574  ; ﾚｰﾝ10上段(M10)切出し上昇
      ORB
      AND     X0  ; 運転準備入り
      AND     M17  ; 運転ﾓｰﾄﾞ
      OUT     M575  ; ﾚｰﾝ10上段(M10)切出し下降
5540  LD      M572  ; ﾚｰﾝ10上段(M10)ﾜｰｸｽﾄｯﾊﾟｰ閉
      ANI     Y159  ; ﾚｰﾝ10上段(M10)ﾜｰｸｽﾄｯﾊﾟｰ開
      OUT     Y158  ; ﾚｰﾝ10上段(M10)ﾜｰｸｽﾄｯﾊﾟｰ閉
5543  LD      M573  ; ﾚｰﾝ10上段(M10)ﾜｰｸｽﾄｯﾊﾟｰ開
      ANI     Y158  ; ﾚｰﾝ10上段(M10)ﾜｰｸｽﾄｯﾊﾟｰ閉
      OUT     Y159  ; ﾚｰﾝ10上段(M10)ﾜｰｸｽﾄｯﾊﾟｰ開
5546  LD      M574  ; ﾚｰﾝ10上段(M10)切出し上昇
      ANI     Y15B  ; ﾚｰﾝ10上段(M10)切出し下降
      OUT     Y15A  ; ﾚｰﾝ10上段(M10)切出し上昇
5549  LD      M575  ; ﾚｰﾝ10上段(M10)切出し下降
      ANI     Y15A  ; ﾚｰﾝ10上段(M10)切出し上昇
      OUT     Y15B  ; ﾚｰﾝ10上段(M10)切出し下降
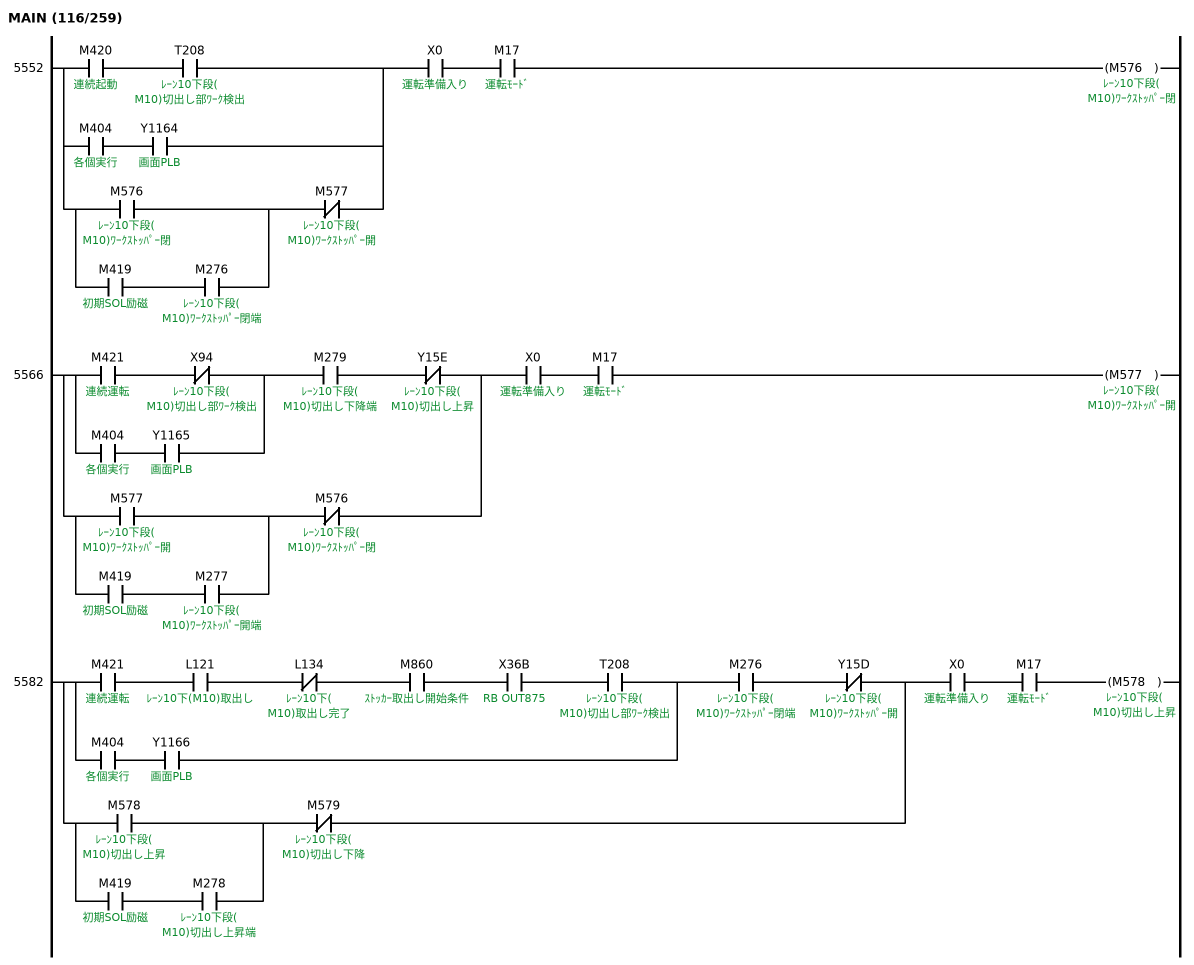
5552  LD      M420  ; 連続起動
      AND     T208  ; ﾚｰﾝ10下段(M10)切出し部ﾜｰｸ検出
      LD      M404  ; 各個実行
      AND     Y1164  ; 画面PLB
      ORB
      LD      M576  ; ﾚｰﾝ10下段(M10)ﾜｰｸｽﾄｯﾊﾟｰ閉
      LD      M419  ; 初期SOL励磁
      AND     M276  ; ﾚｰﾝ10下段(M10)ﾜｰｸｽﾄｯﾊﾟｰ閉端
      ORB
      ANI     M577  ; ﾚｰﾝ10下段(M10)ﾜｰｸｽﾄｯﾊﾟｰ開
      ORB
      AND     X0  ; 運転準備入り
      AND     M17  ; 運転ﾓｰﾄﾞ
      OUT     M576  ; ﾚｰﾝ10下段(M10)ﾜｰｸｽﾄｯﾊﾟｰ閉
5566  LD      M421  ; 連続運転
      ANI     X94  ; ﾚｰﾝ10下段(M10)切出し部ﾜｰｸ検出
      LD      M404  ; 各個実行
      AND     Y1165  ; 画面PLB
      ORB
      AND     M279  ; ﾚｰﾝ10下段(M10)切出し下降端
      ANI     Y15E  ; ﾚｰﾝ10下段(M10)切出し上昇
      LD      M577  ; ﾚｰﾝ10下段(M10)ﾜｰｸｽﾄｯﾊﾟｰ開
      LD      M419  ; 初期SOL励磁
      AND     M277  ; ﾚｰﾝ10下段(M10)ﾜｰｸｽﾄｯﾊﾟｰ開端
      ORB
      ANI     M576  ; ﾚｰﾝ10下段(M10)ﾜｰｸｽﾄｯﾊﾟｰ閉
      ORB
      AND     X0  ; 運転準備入り
      AND     M17  ; 運転ﾓｰﾄﾞ
      OUT     M577  ; ﾚｰﾝ10下段(M10)ﾜｰｸｽﾄｯﾊﾟｰ開
5582  LD      M421  ; 連続運転
      AND     L121  ; ﾚｰﾝ10下(M10)取出し
      ANI     L134  ; ﾚｰﾝ10下(M10)取出し完了
      AND     M860  ; ｽﾄｯｶｰ取出し開始条件
      AND     X36B  ; RB OUT875
      AND     T208  ; ﾚｰﾝ10下段(M10)切出し部ﾜｰｸ検出
      LD      M404  ; 各個実行
      AND     Y1166  ; 画面PLB
      ORB
      AND     M276  ; ﾚｰﾝ10下段(M10)ﾜｰｸｽﾄｯﾊﾟｰ閉端
      ANI     Y15D  ; ﾚｰﾝ10下段(M10)ﾜｰｸｽﾄｯﾊﾟｰ開
      LD      M578  ; ﾚｰﾝ10下段(M10)切出し上昇
      LD      M419  ; 初期SOL励磁
      AND     M278  ; ﾚｰﾝ10下段(M10)切出し上昇端
      ORB
      ANI     M579  ; ﾚｰﾝ10下段(M10)切出し下降
      ORB
      AND     X0  ; 運転準備入り
      AND     M17  ; 運転ﾓｰﾄﾞ
      OUT     M578  ; ﾚｰﾝ10下段(M10)切出し上昇
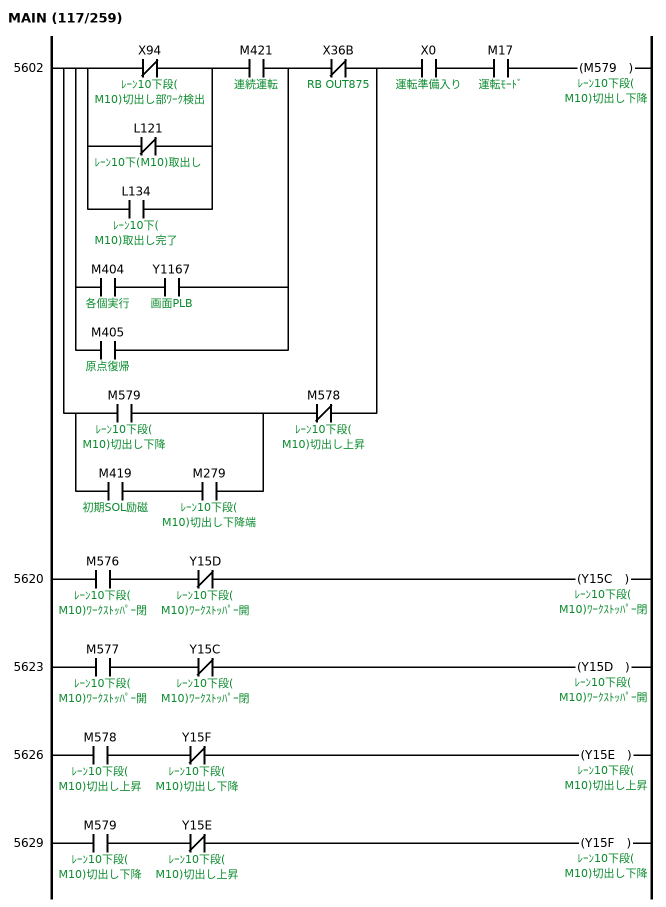
5602  LDI     X94  ; ﾚｰﾝ10下段(M10)切出し部ﾜｰｸ検出
      ORI     L121  ; ﾚｰﾝ10下(M10)取出し
      OR      L134  ; ﾚｰﾝ10下(M10)取出し完了
      AND     M421  ; 連続運転
      LD      M404  ; 各個実行
      AND     Y1167  ; 画面PLB
      ORB
      OR      M405  ; 原点復帰
      ANI     X36B  ; RB OUT875
      LD      M579  ; ﾚｰﾝ10下段(M10)切出し下降
      LD      M419  ; 初期SOL励磁
      AND     M279  ; ﾚｰﾝ10下段(M10)切出し下降端
      ORB
      ANI     M578  ; ﾚｰﾝ10下段(M10)切出し上昇
      ORB
      AND     X0  ; 運転準備入り
      AND     M17  ; 運転ﾓｰﾄﾞ
      OUT     M579  ; ﾚｰﾝ10下段(M10)切出し下降
5620  LD      M576  ; ﾚｰﾝ10下段(M10)ﾜｰｸｽﾄｯﾊﾟｰ閉
      ANI     Y15D  ; ﾚｰﾝ10下段(M10)ﾜｰｸｽﾄｯﾊﾟｰ開
      OUT     Y15C  ; ﾚｰﾝ10下段(M10)ﾜｰｸｽﾄｯﾊﾟｰ閉
5623  LD      M577  ; ﾚｰﾝ10下段(M10)ﾜｰｸｽﾄｯﾊﾟｰ開
      ANI     Y15C  ; ﾚｰﾝ10下段(M10)ﾜｰｸｽﾄｯﾊﾟｰ閉
      OUT     Y15D  ; ﾚｰﾝ10下段(M10)ﾜｰｸｽﾄｯﾊﾟｰ開
5626  LD      M578  ; ﾚｰﾝ10下段(M10)切出し上昇
      ANI     Y15F  ; ﾚｰﾝ10下段(M10)切出し下降
      OUT     Y15E  ; ﾚｰﾝ10下段(M10)切出し上昇
5629  LD      M579  ; ﾚｰﾝ10下段(M10)切出し下降
      ANI     Y15E  ; ﾚｰﾝ10下段(M10)切出し上昇
      OUT     Y15F  ; ﾚｰﾝ10下段(M10)切出し下降
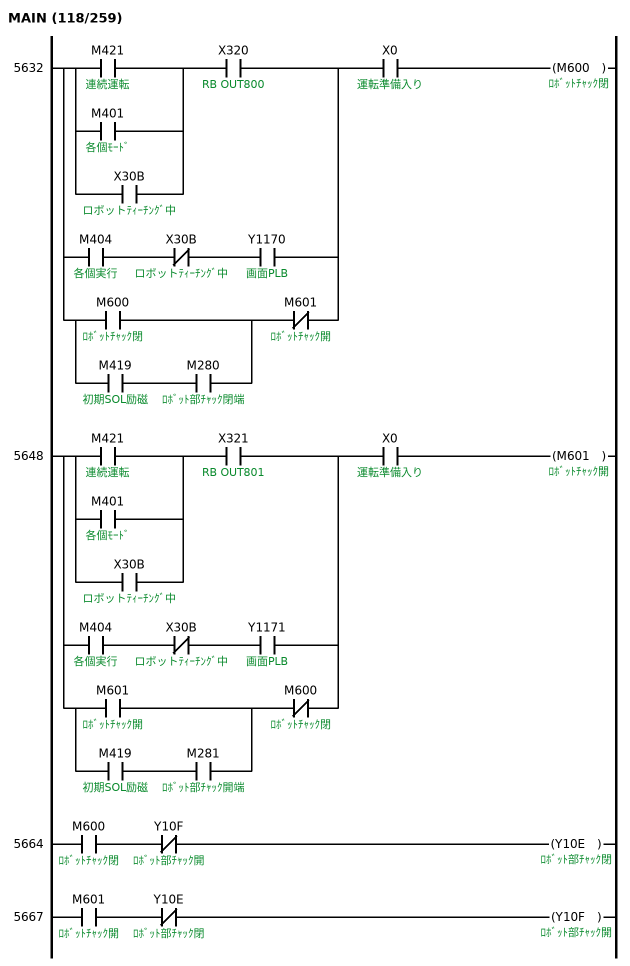
5632  LD      M421  ; 連続運転
      OR      M401  ; 各個ﾓｰﾄﾞ
      OR      X30B  ; ロボットﾃｨｰﾁﾝｸﾞ中
      AND     X320  ; RB OUT800
      LD      M404  ; 各個実行
      ANI     X30B  ; ロボットﾃｨｰﾁﾝｸﾞ中
      AND     Y1170  ; 画面PLB
      ORB
      LD      M600  ; ﾛﾎﾞｯﾄﾁｬｯｸ閉
      LD      M419  ; 初期SOL励磁
      AND     M280  ; ﾛﾎﾞｯﾄ部ﾁｬｯｸ閉端
      ORB
      ANI     M601  ; ﾛﾎﾞｯﾄﾁｬｯｸ開
      ORB
      AND     X0  ; 運転準備入り
      OUT     M600  ; ﾛﾎﾞｯﾄﾁｬｯｸ閉
5648  LD      M421  ; 連続運転
      OR      M401  ; 各個ﾓｰﾄﾞ
      OR      X30B  ; ロボットﾃｨｰﾁﾝｸﾞ中
      AND     X321  ; RB OUT801
      LD      M404  ; 各個実行
      ANI     X30B  ; ロボットﾃｨｰﾁﾝｸﾞ中
      AND     Y1171  ; 画面PLB
      ORB
      LD      M601  ; ﾛﾎﾞｯﾄﾁｬｯｸ開
      LD      M419  ; 初期SOL励磁
      AND     M281  ; ﾛﾎﾞｯﾄ部ﾁｬｯｸ開端
      ORB
      ANI     M600  ; ﾛﾎﾞｯﾄﾁｬｯｸ閉
      ORB
      AND     X0  ; 運転準備入り
      OUT     M601  ; ﾛﾎﾞｯﾄﾁｬｯｸ開
5664  LD      M600  ; ﾛﾎﾞｯﾄﾁｬｯｸ閉
      ANI     Y10F  ; ﾛﾎﾞｯﾄ部ﾁｬｯｸ開
      OUT     Y10E  ; ﾛﾎﾞｯﾄ部ﾁｬｯｸ閉
5667  LD      M601  ; ﾛﾎﾞｯﾄﾁｬｯｸ開
      ANI     Y10E  ; ﾛﾎﾞｯﾄ部ﾁｬｯｸ閉
      OUT     Y10F  ; ﾛﾎﾞｯﾄ部ﾁｬｯｸ開
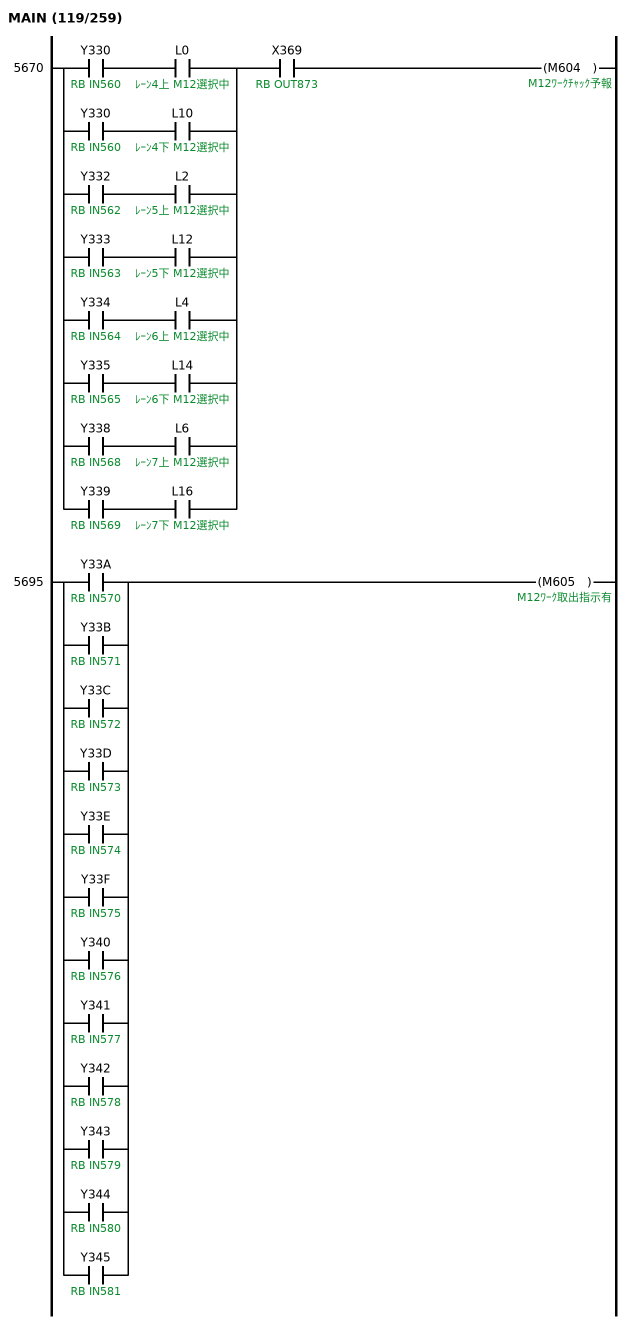
5670  LD      Y330  ; RB IN560
      AND     L0  ; ﾚｰﾝ4上 M12選択中
      LD      Y330  ; RB IN560
      AND     L10  ; ﾚｰﾝ4下 M12選択中
      ORB
      LD      Y332  ; RB IN562
      AND     L2  ; ﾚｰﾝ5上 M12選択中
      ORB
      LD      Y333  ; RB IN563
      AND     L12  ; ﾚｰﾝ5下 M12選択中
      ORB
      LD      Y334  ; RB IN564
      AND     L4  ; ﾚｰﾝ6上 M12選択中
      ORB
      LD      Y335  ; RB IN565
      AND     L14  ; ﾚｰﾝ6下 M12選択中
      ORB
      LD      Y338  ; RB IN568
      AND     L6  ; ﾚｰﾝ7上 M12選択中
      ORB
      LD      Y339  ; RB IN569
      AND     L16  ; ﾚｰﾝ7下 M12選択中
      ORB
      AND     X369  ; RB OUT873
      OUT     M604  ; M12ﾜｰｸﾁｬｯｸ予報
5695  LD      Y33A  ; RB IN570
      OR      Y33B  ; RB IN571
      OR      Y33C  ; RB IN572
      OR      Y33D  ; RB IN573
      OR      Y33E  ; RB IN574
      OR      Y33F  ; RB IN575
      OR      Y340  ; RB IN576
      OR      Y341  ; RB IN577
      OR      Y342  ; RB IN578
      OR      Y343  ; RB IN579
      OR      Y344  ; RB IN580
      OR      Y345  ; RB IN581
      OUT     M605  ; M12ﾜｰｸ取出指示有
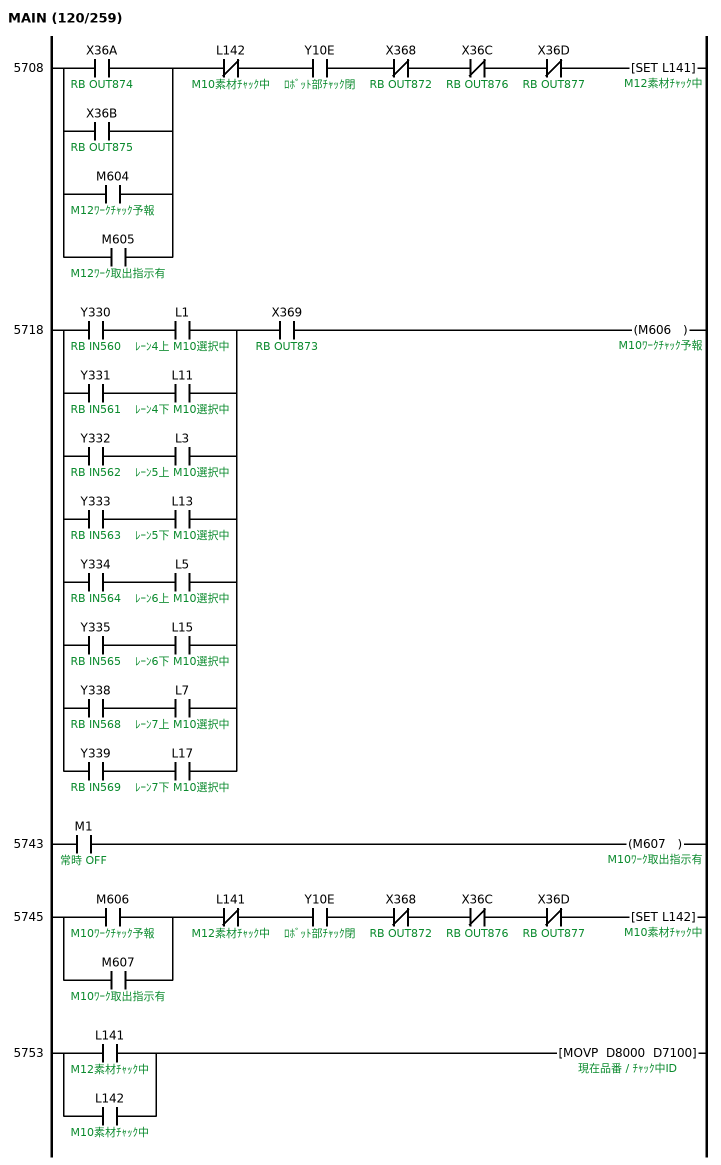
5708  LD      X36A  ; RB OUT874
      OR      X36B  ; RB OUT875
      OR      M604  ; M12ﾜｰｸﾁｬｯｸ予報
      OR      M605  ; M12ﾜｰｸ取出指示有
      ANI     L142  ; M10素材ﾁｬｯｸ中
      AND     Y10E  ; ﾛﾎﾞｯﾄ部ﾁｬｯｸ閉
      ANI     X368  ; RB OUT872
      ANI     X36C  ; RB OUT876
      ANI     X36D  ; RB OUT877
      SET     L141  ; M12素材ﾁｬｯｸ中
5718  LD      Y330  ; RB IN560
      AND     L1  ; ﾚｰﾝ4上 M10選択中
      LD      Y331  ; RB IN561
      AND     L11  ; ﾚｰﾝ4下 M10選択中
      ORB
      LD      Y332  ; RB IN562
      AND     L3  ; ﾚｰﾝ5上 M10選択中
      ORB
      LD      Y333  ; RB IN563
      AND     L13  ; ﾚｰﾝ5下 M10選択中
      ORB
      LD      Y334  ; RB IN564
      AND     L5  ; ﾚｰﾝ6上 M10選択中
      ORB
      LD      Y335  ; RB IN565
      AND     L15  ; ﾚｰﾝ6下 M10選択中
      ORB
      LD      Y338  ; RB IN568
      AND     L7  ; ﾚｰﾝ7上 M10選択中
      ORB
      LD      Y339  ; RB IN569
      AND     L17  ; ﾚｰﾝ7下 M10選択中
      ORB
      AND     X369  ; RB OUT873
      OUT     M606  ; M10ﾜｰｸﾁｬｯｸ予報
5743  LD      M1  ; 常時 OFF
      OUT     M607  ; M10ﾜｰｸ取出指示有
5745  LD      M606  ; M10ﾜｰｸﾁｬｯｸ予報
      OR      M607  ; M10ﾜｰｸ取出指示有
      ANI     L141  ; M12素材ﾁｬｯｸ中
      AND     Y10E  ; ﾛﾎﾞｯﾄ部ﾁｬｯｸ閉
      ANI     X368  ; RB OUT872
      ANI     X36C  ; RB OUT876
      ANI     X36D  ; RB OUT877
      SET     L142  ; M10素材ﾁｬｯｸ中
5753  LD      L141  ; M12素材ﾁｬｯｸ中
      OR      L142  ; M10素材ﾁｬｯｸ中
      MOVP    D8000 D7100  ; 現在品番 / ﾁｬｯｸ中ID
